LIN {X -172.185,Y +1147.423,Z +0.000,A -19.971,E1 -36.175,E3 +84213.761,E4 +0.000} C_DIS
LIN {X -165.999,Y +1152.127,Z +0.000,A -20.000,E1 -32.027,E3 +84233.519,E4 +0.000} C_DIS
LIN {X -160.138,Y +1155.667,Z +0.000,A -20.000,E1 -26.368,E3 +84257.889,E4 +0.000} C_DIS
LIN {X -155.625,Y +1157.756,Z +0.000,A -20.000,E1 -19.505,E3 +84286.565,E4 +0.000} C_DIS
LIN {X -153.552,Y +1158.113,Z +0.000,A -20.000,E1 -11.113,E3 +84322.316,E4 +0.000} C_DIS
LIN {X -156.311,Y +1155.540,Z +0.000,A -20.000,E1 -0.839,E3 +84365.676,E4 +0.000} C_DIS
LIN {X -161.281,Y +1151.851,Z +0.000,A -20.000,E1 +7.737,E3 +84395.575,E4 +0.000} C_DIS
LIN {X -167.493,Y +1147.157,Z +0.000,A -20.000,E1 +16.195,E3 +84420.014,E4 +0.000} C_DIS
LIN {X -173.235,Y +1142.221,Z +0.000,A -20.000,E1 +22.930,E3 +84437.316,E4 +0.000} C_DIS
LIN {X -181.123,Y +1133.734,Z +0.000,A -20.000,E1 +30.868,E3 +84458.072,E4 +0.000} C_DIS
LIN {X -189.654,Y +1120.856,Z +0.000,A -20.000,E1 +39.018,E3 +84480.086,E4 +0.000} C_DIS
LIN {X -195.246,Y +1107.046,Z +0.000,A -20.000,E1 +44.515,E3 +84497.988,E4 +0.000} C_DIS
LIN {X -198.051,Y +1092.368,Z +0.000,A -20.000,E1 +47.947,E3 +84514.514,E4 +0.000} C_DIS
LIN {X -198.143,Y +1081.370,Z +0.000,A -19.806,E1 +49.153,E3 +84526.375,E4 +0.000} C_DIS
LIN {X -197.177,Y +1073.569,Z +0.000,A -17.356,E1 +49.162,E3 +84534.959,E4 +0.000} C_DIS
LIN {X -195.448,Y +1066.139,Z +0.000,A -12.154,E1 +48.512,E3 +84543.554,E4 +0.000} C_DIS
LIN {X -193.346,Y +1058.941,Z +0.000,A -7.133,E1 +47.724,E3 +84552.434,E4 +0.000} C_DIS
LIN {X -191.781,Y +1050.839,Z +0.000,A -3.715,E1 +47.274,E3 +84562.767,E4 +0.000} C_DIS
LIN {X -190.795,Y +1039.355,Z +0.000,A -0.983,E1 +46.842,E3 +84577.427,E4 +0.000} C_DIS
LIN {X -190.395,Y +1028.856,Z +0.000,A -0.089,E1 +46.598,E3 +84590.821,E4 +0.000} C_DIS
LIN {X -190.239,Y +1018.851,Z +0.000,A -0.004,E1 +46.529,E3 +84603.589,E4 +0.000} C_DIS
LIN {X -190.161,Y +1004.975,Z +0.000,A +0.000,E1 +46.506,E3 +84621.303,E4 +0.000} C_DIS
LIN {X -190.142,Y +412.853,Z +0.000,A +0.000,E1 +46.501,E3 +85377.509,E4 +0.000} C_DIS
LIN {X -190.147,Y +401.077,Z +0.000,A +0.000,E1 +46.499,E3 +85392.550,E4 +0.000} C_DIS
LIN {X -190.159,Y +390.929,Z +0.000,A +0.000,E1 +46.494,E3 +85405.516,E4 +0.000} C_DIS
LIN {X -190.174,Y +383.973,Z +0.000,A +0.000,E1 +46.484,E3 +85414.409,E4 +0.000} C_DIS
LIN {X -190.200,Y +373.815,Z +0.000,A +0.000,E1 +46.448,E3 +85427.414,E4 +0.000} C_DIS
LIN {X -190.154,Y +361.003,Z +0.000,A +0.000,E1 +46.303,E3 +85443.908,E4 +0.000} C_DIS
LIN {X -189.772,Y +350.660,Z +0.000,A +0.049,E1 +45.996,E3 +85457.447,E4 +0.000} C_DIS
LIN {X -189.325,Y +346.917,Z +0.000,A +0.243,E1 +45.771,E3 +85462.516,E4 +0.000} C_DIS
LIN {X -188.196,Y +342.754,Z +0.000,A +1.966,E1 +45.249,E3 +85468.524,E4 +0.000} C_DIS
LIN {X -185.199,Y +337.023,Z +0.000,A +6.630,E1 +43.793,E3 +85477.898,E4 +0.000} C_DIS
LIN {X -181.141,Y +331.596,Z +0.000,A +12.274,E1 +41.569,E3 +85488.458,E4 +0.000} C_DIS
LIN {X -176.762,Y +326.804,Z +0.000,A +17.560,E1 +38.898,E3 +85499.882,E4 +0.000} C_DIS
LIN {X -172.184,Y +322.578,Z +0.000,A +19.859,E1 +36.197,E3 +85512.612,E4 +0.000} C_DIS
LIN {X -165.998,Y +317.874,Z +0.000,A +20.000,E1 +32.027,E3 +85532.370,E4 +0.000} C_DIS
LIN {X -160.137,Y +314.334,Z +0.000,A +20.000,E1 +26.368,E3 +85556.739,E4 +0.000} C_DIS
LIN {X -155.624,Y +312.245,Z +0.000,A +20.000,E1 +19.506,E3 +85585.415,E4 +0.000} C_DIS
LIN {X -153.557,Y +311.879,Z +0.000,A +20.000,E1 +11.113,E3 +85621.170,E4 +0.000} C_DIS
LIN {X -155.320,Y +313.348,Z +0.000,A +20.000,E1 +3.401,E3 +85654.354,E4 +0.000} C_DIS
LIN {X -160.005,Y +315.804,Z +0.000,A +20.000,E1 -4.720,E3 +85684.732,E4 +0.000} C_DIS
LIN {X -164.504,Y +318.255,Z +0.000,A +20.000,E1 -10.663,E3 +85704.101,E4 +0.000} C_DIS
LIN {X -170.340,Y +322.684,Z +0.000,A +20.000,E1 -17.457,E3 +85724.133,E4 +0.000} C_DIS
LIN {X -175.568,Y +329.106,Z +0.000,A +20.000,E1 -24.747,E3 +85741.367,E4 +0.000} C_DIS
LIN {X -184.074,Y +340.065,Z +0.000,A +20.000,E1 -33.664,E3 +85764.307,E4 +0.000} C_DIS
LIN {X -190.779,Y +351.388,Z +0.000,A +20.000,E1 -40.083,E3 +85782.085,E4 +0.000} C_DIS
LIN {X -195.254,Y +362.955,Z +0.000,A +20.000,E1 -44.515,E3 +85796.838,E4 +0.000} C_DIS
LIN {X -197.754,Y +374.780,Z +0.000,A +20.000,E1 -47.450,E3 +85810.260,E4 +0.000} C_DIS
LIN {X -198.310,Y +383.215,Z +0.000,A +19.956,E1 -48.698,E3 +85819.384,E4 +0.000} C_DIS
LIN {X -197.912,Y +391.275,Z +0.000,A +18.601,E1 -49.158,E3 +85828.102,E4 +0.000} C_DIS
LIN {X -196.679,Y +398.944,Z +0.000,A +13.989,E1 -48.784,E3 +85836.656,E4 +0.000} C_DIS
LIN {X -194.742,Y +406.288,Z +0.000,A +8.476,E1 -48.001,E3 +85845.339,E4 +0.000} C_DIS
LIN {X -192.748,Y +413.472,Z +0.000,A +3.905,E1 -47.267,E3 +85854.349,E4 +0.000} C_DIS
LIN {X -191.781,Y +419.162,Z +0.000,A +1.739,E1 -46.975,E3 +85861.617,E4 +0.000} C_DIS
LIN {X -190.795,Y +430.646,Z +0.000,A +0.152,E1 -46.707,E3 +85876.278,E4 +0.000} C_DIS
LIN {X -190.395,Y +441.145,Z +0.000,A +0.001,E1 -46.583,E3 +85889.671,E4 +0.000} C_DIS
LIN {X -190.239,Y +451.150,Z +0.000,A -0.000,E1 -46.528,E3 +85902.439,E4 +0.000} C_DIS
LIN {X -190.161,Y +465.026,Z +0.000,A -0.000,E1 -46.506,E3 +85920.154,E4 +0.000} C_DIS
LIN {X -190.142,Y +1057.148,Z +0.000,A -0.000,E1 -46.500,E3 +86676.360,E4 +0.000} C_DIS
LIN {X -190.147,Y +1068.924,Z +0.000,A -0.000,E1 -46.499,E3 +86691.401,E4 +0.000} C_DIS
LIN {X -190.159,Y +1079.072,Z +0.000,A -0.000,E1 -46.493,E3 +86704.366,E4 +0.000} C_DIS
LIN {X -190.174,Y +1086.028,Z +0.000,A -0.000,E1 -46.483,E3 +86713.260,E4 +0.000} C_DIS
LIN {X -190.200,Y +1096.186,Z +0.000,A -0.000,E1 -46.448,E3 +86726.264,E4 +0.000} C_DIS
LIN {X -190.154,Y +1108.998,Z +0.000,A -0.054,E1 -46.295,E3 +86742.759,E4 +0.000} C_DIS
LIN {X -189.772,Y +1119.341,Z +0.000,A -0.752,E1 -45.902,E3 +86756.297,E4 +0.000} C_DIS
LIN {X -189.097,Y +1124.276,Z +0.000,A -2.508,E1 -45.397,E3 +86763.029,E4 +0.000} C_DIS
LIN {X -187.410,Y +1129.069,Z +0.000,A -5.304,E1 -44.585,E3 +86770.202,E4 +0.000} C_DIS
LIN {X -183.899,Y +1134.873,Z +0.000,A -10.372,E1 -42.805,E3 +86780.208,E4 +0.000} C_DIS
LIN {X -179.711,Y +1140.065,Z +0.000,A -15.940,E1 -40.393,E3 +86790.994,E4 +0.000} C_DIS
LIN {X -176.763,Y +1143.197,Z +0.000,A -18.748,E1 -38.674,E3 +86798.732,E4 +0.000} C_DIS
LIN {X -172.185,Y +1147.423,Z +0.000,A -19.971,E1 -36.175,E3 +86811.462,E4 +0.000} C_DIS
LIN {X -165.999,Y +1152.127,Z +0.000,A -20.000,E1 -32.027,E3 +86831.220,E4 +0.000} C_DIS
LIN {X -160.138,Y +1155.667,Z +0.000,A -20.000,E1 -26.368,E3 +86855.590,E4 +0.000} C_DIS
LIN {X -155.625,Y +1157.756,Z +0.000,A -20.000,E1 -19.505,E3 +86884.266,E4 +0.000} C_DIS
LIN {X -153.552,Y +1158.113,Z +0.000,A -20.000,E1 -11.113,E3 +86920.017,E4 +0.000} C_DIS
LIN {X -156.311,Y +1155.540,Z +0.000,A -20.000,E1 -0.839,E3 +86963.377,E4 +0.000} C_DIS
LIN {X -161.281,Y +1151.851,Z +0.000,A -20.000,E1 +7.737,E3 +86993.276,E4 +0.000} C_DIS
LIN {X -167.493,Y +1147.157,Z +0.000,A -20.000,E1 +16.195,E3 +87017.715,E4 +0.000} C_DIS
LIN {X -173.235,Y +1142.221,Z +0.000,A -20.000,E1 +22.930,E3 +87035.017,E4 +0.000} C_DIS
LIN {X -181.123,Y +1133.734,Z +0.000,A -20.000,E1 +30.868,E3 +87055.773,E4 +0.000} C_DIS
LIN {X -189.654,Y +1120.856,Z +0.000,A -20.000,E1 +39.018,E3 +87077.787,E4 +0.000} C_DIS
LIN {X -195.246,Y +1107.046,Z +0.000,A -20.000,E1 +44.515,E3 +87095.689,E4 +0.000} C_DIS
LIN {X -198.051,Y +1092.368,Z +0.000,A -20.000,E1 +47.947,E3 +87112.215,E4 +0.000} C_DIS
LIN {X -198.143,Y +1081.370,Z +0.000,A -19.806,E1 +49.153,E3 +87124.076,E4 +0.000} C_DIS
LIN {X -197.177,Y +1073.569,Z +0.000,A -17.356,E1 +49.162,E3 +87132.660,E4 +0.000} C_DIS
LIN {X -195.448,Y +1066.139,Z +0.000,A -12.154,E1 +48.512,E3 +87141.255,E4 +0.000} C_DIS
LIN {X -193.346,Y +1058.941,Z +0.000,A -7.133,E1 +47.724,E3 +87150.135,E4 +0.000} C_DIS
LIN {X -191.781,Y +1050.839,Z +0.000,A -3.715,E1 +47.274,E3 +87160.468,E4 +0.000} C_DIS
LIN {X -190.795,Y +1039.355,Z +0.000,A -0.983,E1 +46.842,E3 +87175.128,E4 +0.000} C_DIS
LIN {X -190.395,Y +1028.856,Z +0.000,A -0.089,E1 +46.598,E3 +87188.522,E4 +0.000} C_DIS
LIN {X -190.239,Y +1018.851,Z +0.000,A -0.004,E1 +46.529,E3 +87201.290,E4 +0.000} C_DIS
LIN {X -190.161,Y +1004.975,Z +0.000,A +0.000,E1 +46.506,E3 +87219.004,E4 +0.000} C_DIS
LIN {X -190.142,Y +412.853,Z +0.000,A +0.000,E1 +46.501,E3 +87975.210,E4 +0.000} C_DIS
LIN {X -190.147,Y +401.077,Z +0.000,A +0.000,E1 +46.499,E3 +87990.251,E4 +0.000} C_DIS
LIN {X -190.159,Y +390.929,Z +0.000,A +0.000,E1 +46.494,E3 +88003.217,E4 +0.000} C_DIS
LIN {X -190.174,Y +383.973,Z +0.000,A +0.000,E1 +46.484,E3 +88012.110,E4 +0.000} C_DIS
LIN {X -190.200,Y +373.815,Z +0.000,A +0.000,E1 +46.448,E3 +88025.115,E4 +0.000} C_DIS
LIN {X -190.154,Y +361.003,Z +0.000,A +0.000,E1 +46.303,E3 +88041.609,E4 +0.000} C_DIS
LIN {X -189.772,Y +350.660,Z +0.000,A +0.049,E1 +45.996,E3 +88055.148,E4 +0.000} C_DIS
LIN {X -189.325,Y +346.917,Z +0.000,A +0.243,E1 +45.771,E3 +88060.217,E4 +0.000} C_DIS
LIN {X -188.196,Y +342.754,Z +0.000,A +1.966,E1 +45.249,E3 +88066.225,E4 +0.000} C_DIS
LIN {X -185.199,Y +337.023,Z +0.000,A +6.630,E1 +43.793,E3 +88075.599,E4 +0.000} C_DIS
LIN {X -181.141,Y +331.596,Z +0.000,A +12.274,E1 +41.569,E3 +88086.159,E4 +0.000} C_DIS
LIN {X -176.762,Y +326.804,Z +0.000,A +17.560,E1 +38.898,E3 +88097.583,E4 +0.000} C_DIS
LIN {X -172.184,Y +322.578,Z +0.000,A +19.859,E1 +36.197,E3 +88110.313,E4 +0.000} C_DIS
LIN {X -165.998,Y +317.874,Z +0.000,A +20.000,E1 +32.027,E3 +88130.071,E4 +0.000} C_DIS
LIN {X -160.137,Y +314.334,Z +0.000,A +20.000,E1 +26.368,E3 +88154.440,E4 +0.000} C_DIS
LIN {X -155.624,Y +312.245,Z +0.000,A +20.000,E1 +19.506,E3 +88183.116,E4 +0.000} C_DIS
LIN {X -153.557,Y +311.879,Z +0.000,A +20.000,E1 +11.113,E3 +88218.871,E4 +0.000} C_DIS
LIN {X -155.320,Y +313.348,Z +0.000,A +20.000,E1 +3.401,E3 +88252.055,E4 +0.000} C_DIS
LIN {X -160.005,Y +315.804,Z +0.000,A +20.000,E1 -4.720,E3 +88282.433,E4 +0.000} C_DIS
LIN {X -164.504,Y +318.255,Z +0.000,A +20.000,E1 -10.663,E3 +88301.802,E4 +0.000} C_DIS
LIN {X -170.340,Y +322.684,Z +0.000,A +20.000,E1 -17.457,E3 +88321.834,E4 +0.000} C_DIS
LIN {X -175.568,Y +329.106,Z +0.000,A +20.000,E1 -24.747,E3 +88339.068,E4 +0.000} C_DIS
LIN {X -184.074,Y +340.065,Z +0.000,A +20.000,E1 -33.664,E3 +88362.008,E4 +0.000} C_DIS
LIN {X -190.779,Y +351.388,Z +0.000,A +20.000,E1 -40.083,E3 +88379.786,E4 +0.000} C_DIS
LIN {X -195.254,Y +362.955,Z +0.000,A +20.000,E1 -44.515,E3 +88394.539,E4 +0.000} C_DIS
LIN {X -197.754,Y +374.780,Z +0.000,A +20.000,E1 -47.450,E3 +88407.961,E4 +0.000} C_DIS
LIN {X -198.310,Y +383.215,Z +0.000,A +19.956,E1 -48.698,E3 +88417.085,E4 +0.000} C_DIS
LIN {X -197.912,Y +391.275,Z +0.000,A +18.601,E1 -49.158,E3 +88425.803,E4 +0.000} C_DIS
LIN {X -196.679,Y +398.944,Z +0.000,A +13.989,E1 -48.784,E3 +88434.357,E4 +0.000} C_DIS
LIN {X -194.742,Y +406.288,Z +0.000,A +8.476,E1 -48.001,E3 +88443.040,E4 +0.000} C_DIS
LIN {X -192.748,Y +413.472,Z +0.000,A +3.905,E1 -47.267,E3 +88452.050,E4 +0.000} C_DIS
LIN {X -191.781,Y +419.162,Z +0.000,A +1.739,E1 -46.975,E3 +88459.318,E4 +0.000} C_DIS
LIN {X -190.795,Y +430.646,Z +0.000,A +0.152,E1 -46.707,E3 +88473.979,E4 +0.000} C_DIS
LIN {X -190.395,Y +441.145,Z +0.000,A +0.001,E1 -46.583,E3 +88487.372,E4 +0.000} C_DIS
LIN {X -190.239,Y +451.150,Z +0.000,A -0.000,E1 -46.528,E3 +88500.140,E4 +0.000} C_DIS
LIN {X -190.161,Y +465.026,Z +0.000,A -0.000,E1 -46.506,E3 +88517.855,E4 +0.000} C_DIS
LIN {X -190.142,Y +1057.148,Z +0.000,A -0.000,E1 -46.500,E3 +89274.061,E4 +0.000} C_DIS
LIN {X -190.147,Y +1068.924,Z +0.000,A -0.000,E1 -46.499,E3 +89289.102,E4 +0.000} C_DIS
LIN {X -190.159,Y +1079.072,Z +0.000,A -0.000,E1 -46.493,E3 +89302.067,E4 +0.000} C_DIS
LIN {X -190.174,Y +1086.028,Z +0.000,A -0.000,E1 -46.483,E3 +89310.961,E4 +0.000} C_DIS
LIN {X -190.200,Y +1096.186,Z +0.000,A -0.000,E1 -46.448,E3 +89323.965,E4 +0.000} C_DIS
LIN {X -190.154,Y +1108.998,Z +0.000,A -0.054,E1 -46.295,E3 +89340.460,E4 +0.000} C_DIS
LIN {X -189.772,Y +1119.341,Z +0.000,A -0.752,E1 -45.902,E3 +89353.998,E4 +0.000} C_DIS
LIN {X -189.097,Y +1124.276,Z +0.000,A -2.508,E1 -45.397,E3 +89360.730,E4 +0.000} C_DIS
LIN {X -187.410,Y +1129.069,Z +0.000,A -5.304,E1 -44.585,E3 +89367.903,E4 +0.000} C_DIS
LIN {X -183.899,Y +1134.873,Z +0.000,A -10.372,E1 -42.805,E3 +89377.909,E4 +0.000} C_DIS
LIN {X -179.711,Y +1140.065,Z +0.000,A -15.940,E1 -40.393,E3 +89388.695,E4 +0.000} C_DIS
LIN {X -176.763,Y +1143.197,Z +0.000,A -18.748,E1 -38.674,E3 +89396.433,E4 +0.000} C_DIS
LIN {X -172.185,Y +1147.423,Z +0.000,A -19.971,E1 -36.175,E3 +89409.163,E4 +0.000} C_DIS
LIN {X -165.999,Y +1152.127,Z +0.000,A -20.000,E1 -32.027,E3 +89428.921,E4 +0.000} C_DIS
LIN {X -160.138,Y +1155.667,Z +0.000,A -20.000,E1 -26.368,E3 +89453.291,E4 +0.000} C_DIS
LIN {X -155.625,Y +1157.756,Z +0.000,A -20.000,E1 -19.505,E3 +89481.967,E4 +0.000} C_DIS
LIN {X -153.552,Y +1158.113,Z +0.000,A -20.000,E1 -11.113,E3 +89517.718,E4 +0.000} C_DIS
LIN {X -156.311,Y +1155.540,Z +0.000,A -20.000,E1 -0.839,E3 +89561.078,E4 +0.000} C_DIS
LIN {X -161.281,Y +1151.851,Z +0.000,A -20.000,E1 +7.737,E3 +89590.977,E4 +0.000} C_DIS
LIN {X -167.493,Y +1147.157,Z +0.000,A -20.000,E1 +16.195,E3 +89615.416,E4 +0.000} C_DIS
LIN {X -173.235,Y +1142.221,Z +0.000,A -20.000,E1 +22.930,E3 +89632.718,E4 +0.000} C_DIS
LIN {X -181.123,Y +1133.734,Z +0.000,A -20.000,E1 +30.868,E3 +89653.474,E4 +0.000} C_DIS
LIN {X -189.654,Y +1120.856,Z +0.000,A -20.000,E1 +39.018,E3 +89675.488,E4 +0.000} C_DIS
LIN {X -195.246,Y +1107.046,Z +0.000,A -20.000,E1 +44.515,E3 +89693.390,E4 +0.000} C_DIS
LIN {X -198.051,Y +1092.368,Z +0.000,A -20.000,E1 +47.947,E3 +89709.916,E4 +0.000} C_DIS
LIN {X -198.143,Y +1081.370,Z +0.000,A -19.806,E1 +49.153,E3 +89721.777,E4 +0.000} C_DIS
LIN {X -197.177,Y +1073.569,Z +0.000,A -17.356,E1 +49.162,E3 +89730.361,E4 +0.000} C_DIS
LIN {X -195.448,Y +1066.139,Z +0.000,A -12.154,E1 +48.512,E3 +89738.956,E4 +0.000} C_DIS
LIN {X -193.346,Y +1058.941,Z +0.000,A -7.133,E1 +47.724,E3 +89747.836,E4 +0.000} C_DIS
LIN {X -191.781,Y +1050.839,Z +0.000,A -3.715,E1 +47.274,E3 +89758.169,E4 +0.000} C_DIS
LIN {X -190.795,Y +1039.355,Z +0.000,A -0.983,E1 +46.842,E3 +89772.829,E4 +0.000} C_DIS
LIN {X -190.395,Y +1028.856,Z +0.000,A -0.089,E1 +46.598,E3 +89786.223,E4 +0.000} C_DIS
LIN {X -190.239,Y +1018.851,Z +0.000,A -0.004,E1 +46.529,E3 +89798.991,E4 +0.000} C_DIS
LIN {X -190.161,Y +1004.975,Z +0.000,A +0.000,E1 +46.506,E3 +89816.705,E4 +0.000} C_DIS
LIN {X -190.142,Y +412.853,Z +0.000,A +0.000,E1 +46.501,E3 +90572.911,E4 +0.000} C_DIS
LIN {X -190.147,Y +401.077,Z +0.000,A +0.000,E1 +46.499,E3 +90587.952,E4 +0.000} C_DIS
LIN {X -190.159,Y +390.929,Z +0.000,A +0.000,E1 +46.494,E3 +90600.918,E4 +0.000} C_DIS
LIN {X -190.174,Y +383.973,Z +0.000,A +0.000,E1 +46.484,E3 +90609.811,E4 +0.000} C_DIS
LIN {X -190.200,Y +373.815,Z +0.000,A +0.000,E1 +46.448,E3 +90622.816,E4 +0.000} C_DIS
LIN {X -190.154,Y +361.003,Z +0.000,A +0.000,E1 +46.303,E3 +90639.310,E4 +0.000} C_DIS
LIN {X -189.772,Y +350.660,Z +0.000,A +0.049,E1 +45.996,E3 +90652.849,E4 +0.000} C_DIS
LIN {X -189.325,Y +346.917,Z +0.000,A +0.243,E1 +45.771,E3 +90657.918,E4 +0.000} C_DIS
LIN {X -188.196,Y +342.754,Z +0.000,A +1.966,E1 +45.249,E3 +90663.926,E4 +0.000} C_DIS
LIN {X -185.199,Y +337.023,Z +0.000,A +6.630,E1 +43.793,E3 +90673.300,E4 +0.000} C_DIS
LIN {X -181.141,Y +331.596,Z +0.000,A +12.274,E1 +41.569,E3 +90683.860,E4 +0.000} C_DIS
LIN {X -176.762,Y +326.804,Z +0.000,A +17.560,E1 +38.898,E3 +90695.284,E4 +0.000} C_DIS
LIN {X -172.184,Y +322.578,Z +0.000,A +19.859,E1 +36.197,E3 +90708.014,E4 +0.000} C_DIS
LIN {X -165.998,Y +317.874,Z +0.000,A +20.000,E1 +32.027,E3 +90727.772,E4 +0.000} C_DIS
LIN {X -160.137,Y +314.334,Z +0.000,A +20.000,E1 +26.368,E3 +90752.141,E4 +0.000} C_DIS
LIN {X -155.624,Y +312.245,Z +0.000,A +20.000,E1 +19.506,E3 +90780.817,E4 +0.000} C_DIS
LIN {X -153.557,Y +311.879,Z +0.000,A +20.000,E1 +11.113,E3 +90816.572,E4 +0.000} C_DIS
LIN {X -155.320,Y +313.348,Z +0.000,A +20.000,E1 +3.401,E3 +90849.756,E4 +0.000} C_DIS
LIN {X -160.005,Y +315.804,Z +0.000,A +20.000,E1 -4.720,E3 +90880.134,E4 +0.000} C_DIS
LIN {X -164.504,Y +318.255,Z +0.000,A +20.000,E1 -10.663,E3 +90899.503,E4 +0.000} C_DIS
LIN {X -170.340,Y +322.684,Z +0.000,A +20.000,E1 -17.457,E3 +90919.535,E4 +0.000} C_DIS
LIN {X -175.568,Y +329.106,Z +0.000,A +20.000,E1 -24.747,E3 +90936.769,E4 +0.000} C_DIS
LIN {X -184.074,Y +340.065,Z +0.000,A +20.000,E1 -33.664,E3 +90959.709,E4 +0.000} C_DIS
LIN {X -190.779,Y +351.388,Z +0.000,A +20.000,E1 -40.083,E3 +90977.487,E4 +0.000} C_DIS
LIN {X -195.254,Y +362.955,Z +0.000,A +20.000,E1 -44.515,E3 +90992.240,E4 +0.000} C_DIS
LIN {X -197.754,Y +374.780,Z +0.000,A +20.000,E1 -47.450,E3 +91005.662,E4 +0.000} C_DIS
LIN {X -198.310,Y +383.215,Z +0.000,A +19.956,E1 -48.698,E3 +91014.786,E4 +0.000} C_DIS
LIN {X -197.912,Y +391.275,Z +0.000,A +18.601,E1 -49.158,E3 +91023.504,E4 +0.000} C_DIS
LIN {X -196.679,Y +398.944,Z +0.000,A +13.989,E1 -48.784,E3 +91032.058,E4 +0.000} C_DIS
LIN {X -194.742,Y +406.288,Z +0.000,A +8.476,E1 -48.001,E3 +91040.741,E4 +0.000} C_DIS
LIN {X -192.748,Y +413.472,Z +0.000,A +3.905,E1 -47.267,E3 +91049.751,E4 +0.000} C_DIS
LIN {X -191.781,Y +419.162,Z +0.000,A +1.739,E1 -46.975,E3 +91057.019,E4 +0.000} C_DIS
LIN {X -190.795,Y +430.646,Z +0.000,A +0.152,E1 -46.707,E3 +91071.680,E4 +0.000} C_DIS
LIN {X -190.395,Y +441.145,Z +0.000,A +0.001,E1 -46.583,E3 +91085.073,E4 +0.000} C_DIS
LIN {X -190.239,Y +451.150,Z +0.000,A -0.000,E1 -46.528,E3 +91097.841,E4 +0.000} C_DIS
LIN {X -190.161,Y +465.026,Z +0.000,A -0.000,E1 -46.506,E3 +91115.556,E4 +0.000} C_DIS
LIN {X -190.142,Y +1057.148,Z +0.000,A -0.000,E1 -46.500,E3 +91871.762,E4 +0.000} C_DIS
LIN {X -190.147,Y +1068.924,Z +0.000,A -0.000,E1 -46.499,E3 +91886.803,E4 +0.000} C_DIS
LIN {X -190.159,Y +1079.072,Z +0.000,A -0.000,E1 -46.493,E3 +91899.768,E4 +0.000} C_DIS
LIN {X -190.174,Y +1086.028,Z +0.000,A -0.000,E1 -46.483,E3 +91908.662,E4 +0.000} C_DIS
LIN {X -190.200,Y +1096.186,Z +0.000,A -0.000,E1 -46.448,E3 +91921.666,E4 +0.000} C_DIS
LIN {X -190.154,Y +1108.998,Z +0.000,A -0.054,E1 -46.295,E3 +91938.161,E4 +0.000} C_DIS
LIN {X -189.772,Y +1119.341,Z +0.000,A -0.752,E1 -45.902,E3 +91951.699,E4 +0.000} C_DIS
LIN {X -189.097,Y +1124.276,Z +0.000,A -2.508,E1 -45.397,E3 +91958.431,E4 +0.000} C_DIS
LIN {X -187.410,Y +1129.069,Z +0.000,A -5.304,E1 -44.585,E3 +91965.604,E4 +0.000} C_DIS
LIN {X -183.899,Y +1134.873,Z +0.000,A -10.372,E1 -42.805,E3 +91975.610,E4 +0.000} C_DIS
LIN {X -179.711,Y +1140.065,Z +0.000,A -15.940,E1 -40.393,E3 +91986.396,E4 +0.000} C_DIS
LIN {X -176.763,Y +1143.197,Z +0.000,A -18.748,E1 -38.674,E3 +91994.134,E4 +0.000} C_DIS
LIN {X -172.185,Y +1147.423,Z +0.000,A -19.971,E1 -36.175,E3 +92006.864,E4 +0.000} C_DIS
LIN {X -165.999,Y +1152.127,Z +0.000,A -20.000,E1 -32.027,E3 +92026.622,E4 +0.000} C_DIS
LIN {X -160.138,Y +1155.667,Z +0.000,A -20.000,E1 -26.368,E3 +92050.992,E4 +0.000} C_DIS
LIN {X -155.625,Y +1157.756,Z +0.000,A -20.000,E1 -19.505,E3 +92079.668,E4 +0.000} C_DIS
LIN {X -153.552,Y +1158.113,Z +0.000,A -20.000,E1 -11.113,E3 +92115.419,E4 +0.000} C_DIS
LIN {X -156.311,Y +1155.540,Z +0.000,A -20.000,E1 -0.839,E3 +92158.779,E4 +0.000} C_DIS
LIN {X -161.281,Y +1151.851,Z +0.000,A -20.000,E1 +7.737,E3 +92188.678,E4 +0.000} C_DIS
LIN {X -167.493,Y +1147.157,Z +0.000,A -20.000,E1 +16.195,E3 +92213.117,E4 +0.000} C_DIS
LIN {X -173.235,Y +1142.221,Z +0.000,A -20.000,E1 +22.930,E3 +92230.419,E4 +0.000} C_DIS
LIN {X -181.123,Y +1133.734,Z +0.000,A -20.000,E1 +30.868,E3 +92251.175,E4 +0.000} C_DIS
LIN {X -189.654,Y +1120.856,Z +0.000,A -20.000,E1 +39.018,E3 +92273.189,E4 +0.000} C_DIS
LIN {X -195.246,Y +1107.046,Z +0.000,A -20.000,E1 +44.515,E3 +92291.091,E4 +0.000} C_DIS
LIN {X -198.051,Y +1092.368,Z +0.000,A -20.000,E1 +47.947,E3 +92307.617,E4 +0.000} C_DIS
LIN {X -198.143,Y +1081.370,Z +0.000,A -19.806,E1 +49.153,E3 +92319.478,E4 +0.000} C_DIS
LIN {X -197.177,Y +1073.569,Z +0.000,A -17.356,E1 +49.162,E3 +92328.062,E4 +0.000} C_DIS
LIN {X -195.448,Y +1066.139,Z +0.000,A -12.154,E1 +48.512,E3 +92336.657,E4 +0.000} C_DIS
LIN {X -193.346,Y +1058.941,Z +0.000,A -7.133,E1 +47.724,E3 +92345.537,E4 +0.000} C_DIS
LIN {X -191.781,Y +1050.839,Z +0.000,A -3.715,E1 +47.274,E3 +92355.870,E4 +0.000} C_DIS
LIN {X -190.795,Y +1039.355,Z +0.000,A -0.983,E1 +46.842,E3 +92370.530,E4 +0.000} C_DIS
LIN {X -190.395,Y +1028.856,Z +0.000,A -0.089,E1 +46.598,E3 +92383.924,E4 +0.000} C_DIS
LIN {X -190.239,Y +1018.851,Z +0.000,A -0.004,E1 +46.529,E3 +92396.692,E4 +0.000} C_DIS
LIN {X -190.161,Y +1004.975,Z +0.000,A +0.000,E1 +46.506,E3 +92414.406,E4 +0.000} C_DIS
LIN {X -190.142,Y +412.853,Z +0.000,A +0.000,E1 +46.501,E3 +93170.612,E4 +0.000} C_DIS
LIN {X -190.147,Y +401.077,Z +0.000,A +0.000,E1 +46.499,E3 +93185.653,E4 +0.000} C_DIS
LIN {X -190.159,Y +390.929,Z +0.000,A +0.000,E1 +46.494,E3 +93198.619,E4 +0.000} C_DIS
LIN {X -190.174,Y +383.973,Z +0.000,A +0.000,E1 +46.484,E3 +93207.512,E4 +0.000} C_DIS
LIN {X -190.200,Y +373.815,Z +0.000,A +0.000,E1 +46.448,E3 +93220.517,E4 +0.000} C_DIS
LIN {X -190.154,Y +361.003,Z +0.000,A +0.000,E1 +46.303,E3 +93237.011,E4 +0.000} C_DIS
LIN {X -189.772,Y +350.660,Z +0.000,A +0.049,E1 +45.996,E3 +93250.550,E4 +0.000} C_DIS
LIN {X -189.325,Y +346.917,Z +0.000,A +0.243,E1 +45.771,E3 +93255.619,E4 +0.000} C_DIS
LIN {X -188.196,Y +342.754,Z +0.000,A +1.966,E1 +45.249,E3 +93261.627,E4 +0.000} C_DIS
LIN {X -185.199,Y +337.023,Z +0.000,A +6.630,E1 +43.793,E3 +93271.001,E4 +0.000} C_DIS
LIN {X -181.141,Y +331.596,Z +0.000,A +12.274,E1 +41.569,E3 +93281.561,E4 +0.000} C_DIS
LIN {X -176.762,Y +326.804,Z +0.000,A +17.560,E1 +38.898,E3 +93292.985,E4 +0.000} C_DIS
LIN {X -172.184,Y +322.578,Z +0.000,A +19.859,E1 +36.197,E3 +93305.715,E4 +0.000} C_DIS
LIN {X -165.998,Y +317.874,Z +0.000,A +20.000,E1 +32.027,E3 +93325.473,E4 +0.000} C_DIS
LIN {X -160.137,Y +314.334,Z +0.000,A +20.000,E1 +26.368,E3 +93349.842,E4 +0.000} C_DIS
LIN {X -155.624,Y +312.245,Z +0.000,A +20.000,E1 +19.506,E3 +93378.518,E4 +0.000} C_DIS
LIN {X -153.557,Y +311.879,Z +0.000,A +20.000,E1 +11.113,E3 +93414.273,E4 +0.000} C_DIS
LIN {X -155.320,Y +313.348,Z +0.000,A +20.000,E1 +3.401,E3 +93447.457,E4 +0.000} C_DIS
LIN {X -160.005,Y +315.804,Z +0.000,A +20.000,E1 -4.720,E3 +93477.835,E4 +0.000} C_DIS
LIN {X -164.504,Y +318.255,Z +0.000,A +20.000,E1 -10.663,E3 +93497.204,E4 +0.000} C_DIS
LIN {X -170.340,Y +322.684,Z +0.000,A +20.000,E1 -17.457,E3 +93517.236,E4 +0.000} C_DIS
LIN {X -175.568,Y +329.106,Z +0.000,A +20.000,E1 -24.747,E3 +93534.470,E4 +0.000} C_DIS
LIN {X -184.074,Y +340.065,Z +0.000,A +20.000,E1 -33.664,E3 +93557.410,E4 +0.000} C_DIS
LIN {X -190.779,Y +351.388,Z +0.000,A +20.000,E1 -40.083,E3 +93575.188,E4 +0.000} C_DIS
LIN {X -195.254,Y +362.955,Z +0.000,A +20.000,E1 -44.515,E3 +93589.941,E4 +0.000} C_DIS
LIN {X -197.754,Y +374.780,Z +0.000,A +20.000,E1 -47.450,E3 +93603.363,E4 +0.000} C_DIS
LIN {X -198.310,Y +383.215,Z +0.000,A +19.956,E1 -48.698,E3 +93612.487,E4 +0.000} C_DIS
LIN {X -197.912,Y +391.275,Z +0.000,A +18.601,E1 -49.158,E3 +93621.205,E4 +0.000} C_DIS
LIN {X -196.679,Y +398.944,Z +0.000,A +13.989,E1 -48.784,E3 +93629.759,E4 +0.000} C_DIS
LIN {X -194.742,Y +406.288,Z +0.000,A +8.476,E1 -48.001,E3 +93638.442,E4 +0.000} C_DIS
LIN {X -192.748,Y +413.472,Z +0.000,A +3.905,E1 -47.267,E3 +93647.452,E4 +0.000} C_DIS
LIN {X -191.781,Y +419.162,Z +0.000,A +1.739,E1 -46.975,E3 +93654.720,E4 +0.000} C_DIS
LIN {X -190.795,Y +430.646,Z +0.000,A +0.152,E1 -46.707,E3 +93669.381,E4 +0.000} C_DIS
LIN {X -190.395,Y +441.145,Z +0.000,A +0.001,E1 -46.583,E3 +93682.774,E4 +0.000} C_DIS
LIN {X -190.239,Y +451.150,Z +0.000,A -0.000,E1 -46.528,E3 +93695.542,E4 +0.000} C_DIS
LIN {X -190.161,Y +465.026,Z +0.000,A -0.000,E1 -46.506,E3 +93713.257,E4 +0.000} C_DIS
LIN {X -190.142,Y +1057.148,Z +0.000,A -0.000,E1 -46.500,E3 +94469.463,E4 +0.000} C_DIS
LIN {X -190.147,Y +1068.924,Z +0.000,A -0.000,E1 -46.499,E3 +94484.504,E4 +0.000} C_DIS
LIN {X -190.159,Y +1079.072,Z +0.000,A -0.000,E1 -46.493,E3 +94497.469,E4 +0.000} C_DIS
LIN {X -190.174,Y +1086.028,Z +0.000,A -0.000,E1 -46.483,E3 +94506.363,E4 +0.000} C_DIS
LIN {X -190.200,Y +1096.186,Z +0.000,A -0.000,E1 -46.448,E3 +94519.367,E4 +0.000} C_DIS
LIN {X -190.154,Y +1108.998,Z +0.000,A -0.054,E1 -46.295,E3 +94535.862,E4 +0.000} C_DIS
LIN {X -189.772,Y +1119.341,Z +0.000,A -0.752,E1 -45.902,E3 +94549.400,E4 +0.000} C_DIS
LIN {X -189.097,Y +1124.276,Z +0.000,A -2.508,E1 -45.397,E3 +94556.132,E4 +0.000} C_DIS
LIN {X -187.410,Y +1129.069,Z +0.000,A -5.304,E1 -44.585,E3 +94563.305,E4 +0.000} C_DIS
LIN {X -183.899,Y +1134.873,Z +0.000,A -10.372,E1 -42.805,E3 +94573.311,E4 +0.000} C_DIS
LIN {X -179.711,Y +1140.065,Z +0.000,A -15.940,E1 -40.393,E3 +94584.097,E4 +0.000} C_DIS
LIN {X -176.763,Y +1143.197,Z +0.000,A -18.748,E1 -38.674,E3 +94591.835,E4 +0.000} C_DIS
LIN {X -172.185,Y +1147.423,Z +0.000,A -19.971,E1 -36.175,E3 +94604.565,E4 +0.000} C_DIS
LIN {X -165.999,Y +1152.127,Z +0.000,A -20.000,E1 -32.027,E3 +94624.323,E4 +0.000} C_DIS
LIN {X -160.138,Y +1155.667,Z +0.000,A -20.000,E1 -26.368,E3 +94648.693,E4 +0.000} C_DIS
LIN {X -155.625,Y +1157.756,Z +0.000,A -20.000,E1 -19.505,E3 +94677.369,E4 +0.000} C_DIS
LIN {X -153.552,Y +1158.113,Z +0.000,A -20.000,E1 -11.113,E3 +94713.120,E4 +0.000} C_DIS
LIN {X -156.311,Y +1155.540,Z +0.000,A -20.000,E1 -0.839,E3 +94756.480,E4 +0.000} C_DIS
LIN {X -161.281,Y +1151.851,Z +0.000,A -20.000,E1 +7.737,E3 +94786.379,E4 +0.000} C_DIS
LIN {X -167.493,Y +1147.157,Z +0.000,A -20.000,E1 +16.195,E3 +94810.818,E4 +0.000} C_DIS
LIN {X -173.235,Y +1142.221,Z +0.000,A -20.000,E1 +22.930,E3 +94828.120,E4 +0.000} C_DIS
LIN {X -181.123,Y +1133.734,Z +0.000,A -20.000,E1 +30.868,E3 +94848.876,E4 +0.000} C_DIS
LIN {X -189.654,Y +1120.856,Z +0.000,A -20.000,E1 +39.018,E3 +94870.890,E4 +0.000} C_DIS
LIN {X -195.246,Y +1107.046,Z +0.000,A -20.000,E1 +44.515,E3 +94888.792,E4 +0.000} C_DIS
LIN {X -198.051,Y +1092.368,Z +0.000,A -20.000,E1 +47.947,E3 +94905.318,E4 +0.000} C_DIS
LIN {X -198.143,Y +1081.370,Z +0.000,A -19.806,E1 +49.153,E3 +94917.179,E4 +0.000} C_DIS
LIN {X -197.177,Y +1073.569,Z +0.000,A -17.356,E1 +49.162,E3 +94925.763,E4 +0.000} C_DIS
LIN {X -195.448,Y +1066.139,Z +0.000,A -12.154,E1 +48.512,E3 +94934.358,E4 +0.000} C_DIS
LIN {X -193.346,Y +1058.941,Z +0.000,A -7.133,E1 +47.724,E3 +94943.238,E4 +0.000} C_DIS
LIN {X -191.781,Y +1050.839,Z +0.000,A -3.715,E1 +47.274,E3 +94953.571,E4 +0.000} C_DIS
LIN {X -190.795,Y +1039.355,Z +0.000,A -0.983,E1 +46.842,E3 +94968.231,E4 +0.000} C_DIS
LIN {X -190.395,Y +1028.856,Z +0.000,A -0.089,E1 +46.598,E3 +94981.625,E4 +0.000} C_DIS
LIN {X -190.239,Y +1018.851,Z +0.000,A -0.004,E1 +46.529,E3 +94994.393,E4 +0.000} C_DIS
LIN {X -190.161,Y +1004.975,Z +0.000,A +0.000,E1 +46.506,E3 +95012.107,E4 +0.000} C_DIS
LIN {X -190.142,Y +412.853,Z +0.000,A +0.000,E1 +46.501,E3 +95768.313,E4 +0.000} C_DIS
LIN {X -190.147,Y +401.077,Z +0.000,A +0.000,E1 +46.499,E3 +95783.354,E4 +0.000} C_DIS
LIN {X -190.159,Y +390.929,Z +0.000,A +0.000,E1 +46.494,E3 +95796.320,E4 +0.000} C_DIS
LIN {X -190.174,Y +383.973,Z +0.000,A +0.000,E1 +46.484,E3 +95805.213,E4 +0.000} C_DIS
LIN {X -190.200,Y +373.815,Z +0.000,A +0.000,E1 +46.448,E3 +95818.218,E4 +0.000} C_DIS
LIN {X -190.154,Y +361.003,Z +0.000,A +0.000,E1 +46.303,E3 +95834.712,E4 +0.000} C_DIS
LIN {X -189.772,Y +350.660,Z +0.000,A +0.049,E1 +45.996,E3 +95848.251,E4 +0.000} C_DIS
LIN {X -189.325,Y +346.917,Z +0.000,A +0.243,E1 +45.771,E3 +95853.320,E4 +0.000} C_DIS
LIN {X -188.196,Y +342.754,Z +0.000,A +1.966,E1 +45.249,E3 +95859.328,E4 +0.000} C_DIS
LIN {X -185.199,Y +337.023,Z +0.000,A +6.630,E1 +43.793,E3 +95868.702,E4 +0.000} C_DIS
LIN {X -181.141,Y +331.596,Z +0.000,A +12.274,E1 +41.569,E3 +95879.262,E4 +0.000} C_DIS
LIN {X -176.762,Y +326.804,Z +0.000,A +17.560,E1 +38.898,E3 +95890.686,E4 +0.000} C_DIS
LIN {X -172.184,Y +322.578,Z +0.000,A +19.859,E1 +36.197,E3 +95903.416,E4 +0.000} C_DIS
LIN {X -165.998,Y +317.874,Z +0.000,A +20.000,E1 +32.027,E3 +95923.174,E4 +0.000} C_DIS
LIN {X -160.137,Y +314.334,Z +0.000,A +20.000,E1 +26.368,E3 +95947.543,E4 +0.000} C_DIS
LIN {X -155.624,Y +312.245,Z +0.000,A +20.000,E1 +19.506,E3 +95976.219,E4 +0.000} C_DIS
LIN {X -153.557,Y +311.879,Z +0.000,A +20.000,E1 +11.113,E3 +96011.974,E4 +0.000} C_DIS
LIN {X -155.320,Y +313.348,Z +0.000,A +20.000,E1 +3.401,E3 +96045.158,E4 +0.000} C_DIS
LIN {X -160.005,Y +315.804,Z +0.000,A +20.000,E1 -4.720,E3 +96075.536,E4 +0.000} C_DIS
LIN {X -164.504,Y +318.255,Z +0.000,A +20.000,E1 -10.663,E3 +96094.905,E4 +0.000} C_DIS
LIN {X -170.340,Y +322.684,Z +0.000,A +20.000,E1 -17.457,E3 +96114.937,E4 +0.000} C_DIS
LIN {X -175.568,Y +329.106,Z +0.000,A +20.000,E1 -24.747,E3 +96132.171,E4 +0.000} C_DIS
LIN {X -184.074,Y +340.065,Z +0.000,A +20.000,E1 -33.664,E3 +96155.111,E4 +0.000} C_DIS
LIN {X -190.779,Y +351.388,Z +0.000,A +20.000,E1 -40.083,E3 +96172.889,E4 +0.000} C_DIS
LIN {X -195.254,Y +362.955,Z +0.000,A +20.000,E1 -44.515,E3 +96187.642,E4 +0.000} C_DIS
LIN {X -197.754,Y +374.780,Z +0.000,A +20.000,E1 -47.450,E3 +96201.064,E4 +0.000} C_DIS
LIN {X -198.310,Y +383.215,Z +0.000,A +19.956,E1 -48.698,E3 +96210.188,E4 +0.000} C_DIS
LIN {X -197.912,Y +391.275,Z +0.000,A +18.601,E1 -49.158,E3 +96218.906,E4 +0.000} C_DIS
LIN {X -196.679,Y +398.944,Z +0.000,A +13.989,E1 -48.784,E3 +96227.460,E4 +0.000} C_DIS
LIN {X -194.742,Y +406.288,Z +0.000,A +8.476,E1 -48.001,E3 +96236.143,E4 +0.000} C_DIS
LIN {X -192.748,Y +413.472,Z +0.000,A +3.905,E1 -47.267,E3 +96245.153,E4 +0.000} C_DIS
LIN {X -191.781,Y +419.162,Z +0.000,A +1.739,E1 -46.975,E3 +96252.421,E4 +0.000} C_DIS
LIN {X -190.795,Y +430.646,Z +0.000,A +0.152,E1 -46.707,E3 +96267.082,E4 +0.000} C_DIS
LIN {X -190.395,Y +441.145,Z +0.000,A +0.001,E1 -46.583,E3 +96280.475,E4 +0.000} C_DIS
LIN {X -190.239,Y +451.150,Z +0.000,A -0.000,E1 -46.528,E3 +96293.243,E4 +0.000} C_DIS
LIN {X -190.161,Y +465.026,Z +0.000,A -0.000,E1 -46.506,E3 +96310.958,E4 +0.000} C_DIS
LIN {X -190.142,Y +1057.148,Z +0.000,A -0.000,E1 -46.500,E3 +97067.164,E4 +0.000} C_DIS
LIN {X -190.147,Y +1068.924,Z +0.000,A -0.000,E1 -46.499,E3 +97082.205,E4 +0.000} C_DIS
LIN {X -190.159,Y +1079.072,Z +0.000,A -0.000,E1 -46.493,E3 +97095.170,E4 +0.000} C_DIS
LIN {X -190.174,Y +1086.028,Z +0.000,A -0.000,E1 -46.483,E3 +97104.064,E4 +0.000} C_DIS
LIN {X -190.200,Y +1096.186,Z +0.000,A -0.000,E1 -46.448,E3 +97117.068,E4 +0.000} C_DIS
LIN {X -190.154,Y +1108.998,Z +0.000,A -0.054,E1 -46.295,E3 +97133.563,E4 +0.000} C_DIS
LIN {X -189.772,Y +1119.341,Z +0.000,A -0.752,E1 -45.902,E3 +97147.101,E4 +0.000} C_DIS
LIN {X -189.097,Y +1124.276,Z +0.000,A -2.508,E1 -45.397,E3 +97153.833,E4 +0.000} C_DIS
LIN {X -187.410,Y +1129.069,Z +0.000,A -5.304,E1 -44.585,E3 +97161.006,E4 +0.000} C_DIS
LIN {X -183.899,Y +1134.873,Z +0.000,A -10.372,E1 -42.805,E3 +97171.012,E4 +0.000} C_DIS
LIN {X -179.711,Y +1140.065,Z +0.000,A -15.940,E1 -40.393,E3 +97181.798,E4 +0.000} C_DIS
LIN {X -176.763,Y +1143.197,Z +0.000,A -18.748,E1 -38.674,E3 +97189.536,E4 +0.000} C_DIS
LIN {X -172.185,Y +1147.423,Z +0.000,A -19.971,E1 -36.175,E3 +97202.266,E4 +0.000} C_DIS
LIN {X -165.999,Y +1152.127,Z +0.000,A -20.000,E1 -32.027,E3 +97222.024,E4 +0.000} C_DIS
LIN {X -160.138,Y +1155.667,Z +0.000,A -20.000,E1 -26.368,E3 +97246.394,E4 +0.000} C_DIS
LIN {X -155.625,Y +1157.756,Z +0.000,A -20.000,E1 -19.505,E3 +97275.070,E4 +0.000} C_DIS
LIN {X -153.552,Y +1158.113,Z +0.000,A -20.000,E1 -11.113,E3 +97310.821,E4 +0.000} C_DIS
LIN {X -156.311,Y +1155.540,Z +0.000,A -20.000,E1 -0.839,E3 +97354.181,E4 +0.000} C_DIS
LIN {X -161.281,Y +1151.851,Z +0.000,A -20.000,E1 +7.737,E3 +97384.080,E4 +0.000} C_DIS
LIN {X -167.493,Y +1147.157,Z +0.000,A -20.000,E1 +16.195,E3 +97408.519,E4 +0.000} C_DIS
LIN {X -173.235,Y +1142.221,Z +0.000,A -20.000,E1 +22.930,E3 +97425.821,E4 +0.000} C_DIS
LIN {X -181.123,Y +1133.734,Z +0.000,A -20.000,E1 +30.868,E3 +97446.577,E4 +0.000} C_DIS
LIN {X -189.654,Y +1120.856,Z +0.000,A -20.000,E1 +39.018,E3 +97468.591,E4 +0.000} C_DIS
LIN {X -195.246,Y +1107.046,Z +0.000,A -20.000,E1 +44.515,E3 +97486.493,E4 +0.000} C_DIS
LIN {X -198.051,Y +1092.368,Z +0.000,A -20.000,E1 +47.947,E3 +97503.019,E4 +0.000} C_DIS
LIN {X -198.143,Y +1081.370,Z +0.000,A -19.806,E1 +49.153,E3 +97514.880,E4 +0.000} C_DIS
LIN {X -197.177,Y +1073.569,Z +0.000,A -17.356,E1 +49.162,E3 +97523.464,E4 +0.000} C_DIS
LIN {X -195.448,Y +1066.139,Z +0.000,A -12.154,E1 +48.512,E3 +97532.059,E4 +0.000} C_DIS
LIN {X -193.346,Y +1058.941,Z +0.000,A -7.133,E1 +47.724,E3 +97540.939,E4 +0.000} C_DIS
LIN {X -191.781,Y +1050.839,Z +0.000,A -3.715,E1 +47.274,E3 +97551.272,E4 +0.000} C_DIS
LIN {X -190.795,Y +1039.355,Z +0.000,A -0.983,E1 +46.842,E3 +97565.932,E4 +0.000} C_DIS
LIN {X -190.395,Y +1028.856,Z +0.000,A -0.089,E1 +46.598,E3 +97579.326,E4 +0.000} C_DIS
LIN {X -190.239,Y +1018.851,Z +0.000,A -0.004,E1 +46.529,E3 +97592.094,E4 +0.000} C_DIS
LIN {X -190.161,Y +1004.975,Z +0.000,A +0.000,E1 +46.506,E3 +97609.808,E4 +0.000} C_DIS
LIN {X -190.142,Y +412.853,Z +0.000,A +0.000,E1 +46.501,E3 +98366.014,E4 +0.000} C_DIS
LIN {X -190.147,Y +401.077,Z +0.000,A +0.000,E1 +46.499,E3 +98381.055,E4 +0.000} C_DIS
LIN {X -190.159,Y +390.929,Z +0.000,A +0.000,E1 +46.494,E3 +98394.021,E4 +0.000} C_DIS
LIN {X -190.174,Y +383.973,Z +0.000,A +0.000,E1 +46.484,E3 +98402.914,E4 +0.000} C_DIS
LIN {X -190.200,Y +373.815,Z +0.000,A +0.000,E1 +46.448,E3 +98415.919,E4 +0.000} C_DIS
LIN {X -190.154,Y +361.003,Z +0.000,A +0.000,E1 +46.303,E3 +98432.413,E4 +0.000} C_DIS
LIN {X -189.772,Y +350.660,Z +0.000,A +0.049,E1 +45.996,E3 +98445.952,E4 +0.000} C_DIS
LIN {X -189.325,Y +346.917,Z +0.000,A +0.243,E1 +45.771,E3 +98451.021,E4 +0.000} C_DIS
LIN {X -188.196,Y +342.754,Z +0.000,A +1.966,E1 +45.249,E3 +98457.029,E4 +0.000} C_DIS
LIN {X -185.199,Y +337.023,Z +0.000,A +6.630,E1 +43.793,E3 +98466.403,E4 +0.000} C_DIS
LIN {X -181.141,Y +331.596,Z +0.000,A +12.274,E1 +41.569,E3 +98476.963,E4 +0.000} C_DIS
LIN {X -176.762,Y +326.804,Z +0.000,A +17.560,E1 +38.898,E3 +98488.387,E4 +0.000} C_DIS
LIN {X -172.184,Y +322.578,Z +0.000,A +19.859,E1 +36.197,E3 +98501.117,E4 +0.000} C_DIS
LIN {X -165.998,Y +317.874,Z +0.000,A +20.000,E1 +32.027,E3 +98520.875,E4 +0.000} C_DIS
LIN {X -160.137,Y +314.334,Z +0.000,A +20.000,E1 +26.368,E3 +98545.244,E4 +0.000} C_DIS
LIN {X -155.624,Y +312.245,Z +0.000,A +20.000,E1 +19.506,E3 +98573.920,E4 +0.000} C_DIS
LIN {X -153.557,Y +311.879,Z +0.000,A +20.000,E1 +11.113,E3 +98609.675,E4 +0.000} C_DIS
LIN {X -155.320,Y +313.348,Z +0.000,A +20.000,E1 +3.401,E3 +98642.859,E4 +0.000} C_DIS
LIN {X -160.005,Y +315.804,Z +0.000,A +20.000,E1 -4.720,E3 +98673.237,E4 +0.000} C_DIS
LIN {X -164.504,Y +318.255,Z +0.000,A +20.000,E1 -10.663,E3 +98692.606,E4 +0.000} C_DIS
LIN {X -170.340,Y +322.684,Z +0.000,A +20.000,E1 -17.457,E3 +98712.638,E4 +0.000} C_DIS
LIN {X -175.568,Y +329.106,Z +0.000,A +20.000,E1 -24.747,E3 +98729.872,E4 +0.000} C_DIS
LIN {X -184.074,Y +340.065,Z +0.000,A +20.000,E1 -33.664,E3 +98752.812,E4 +0.000} C_DIS
LIN {X -190.779,Y +351.388,Z +0.000,A +20.000,E1 -40.083,E3 +98770.590,E4 +0.000} C_DIS
LIN {X -195.254,Y +362.955,Z +0.000,A +20.000,E1 -44.515,E3 +98785.343,E4 +0.000} C_DIS
LIN {X -197.754,Y +374.780,Z +0.000,A +20.000,E1 -47.450,E3 +98798.765,E4 +0.000} C_DIS
LIN {X -198.310,Y +383.215,Z +0.000,A +19.956,E1 -48.698,E3 +98807.889,E4 +0.000} C_DIS
LIN {X -197.912,Y +391.275,Z +0.000,A +18.601,E1 -49.158,E3 +98816.607,E4 +0.000} C_DIS
LIN {X -196.679,Y +398.944,Z +0.000,A +13.989,E1 -48.784,E3 +98825.161,E4 +0.000} C_DIS
LIN {X -194.742,Y +406.288,Z +0.000,A +8.476,E1 -48.001,E3 +98833.844,E4 +0.000} C_DIS
LIN {X -192.748,Y +413.472,Z +0.000,A +3.905,E1 -47.267,E3 +98842.854,E4 +0.000} C_DIS
LIN {X -191.781,Y +419.162,Z +0.000,A +1.739,E1 -46.975,E3 +98850.122,E4 +0.000} C_DIS
LIN {X -190.795,Y +430.646,Z +0.000,A +0.152,E1 -46.707,E3 +98864.783,E4 +0.000} C_DIS
LIN {X -190.395,Y +441.145,Z +0.000,A +0.001,E1 -46.583,E3 +98878.176,E4 +0.000} C_DIS
LIN {X -190.239,Y +451.150,Z +0.000,A -0.000,E1 -46.528,E3 +98890.944,E4 +0.000} C_DIS
LIN {X -190.161,Y +465.026,Z +0.000,A -0.000,E1 -46.506,E3 +98908.659,E4 +0.000} C_DIS
LIN {X -190.142,Y +1057.148,Z +0.000,A -0.000,E1 -46.500,E3 +99664.865,E4 +0.000} C_DIS
LIN {X -190.147,Y +1068.924,Z +0.000,A -0.000,E1 -46.499,E3 +99679.906,E4 +0.000} C_DIS
LIN {X -190.159,Y +1079.072,Z +0.000,A -0.000,E1 -46.493,E3 +99692.871,E4 +0.000} C_DIS
LIN {X -190.174,Y +1086.028,Z +0.000,A -0.000,E1 -46.483,E3 +99701.765,E4 +0.000} C_DIS
LIN {X -190.200,Y +1096.186,Z +0.000,A -0.000,E1 -46.448,E3 +99714.769,E4 +0.000} C_DIS
LIN {X -190.154,Y +1108.998,Z +0.000,A -0.054,E1 -46.295,E3 +99731.264,E4 +0.000} C_DIS
LIN {X -189.772,Y +1119.341,Z +0.000,A -0.752,E1 -45.902,E3 +99744.802,E4 +0.000} C_DIS
LIN {X -189.097,Y +1124.276,Z +0.000,A -2.508,E1 -45.397,E3 +99751.534,E4 +0.000} C_DIS
LIN {X -187.410,Y +1129.069,Z +0.000,A -5.304,E1 -44.585,E3 +99758.707,E4 +0.000} C_DIS
LIN {X -183.899,Y +1134.873,Z +0.000,A -10.372,E1 -42.805,E3 +99768.713,E4 +0.000} C_DIS
LIN {X -179.711,Y +1140.065,Z +0.000,A -15.940,E1 -40.393,E3 +99779.499,E4 +0.000} C_DIS
LIN {X -176.763,Y +1143.197,Z +0.000,A -18.748,E1 -38.674,E3 +99787.237,E4 +0.000} C_DIS
LIN {X -172.185,Y +1147.423,Z +0.000,A -19.971,E1 -36.175,E3 +99799.967,E4 +0.000} C_DIS
LIN {X -165.999,Y +1152.127,Z +0.000,A -20.000,E1 -32.027,E3 +99819.725,E4 +0.000} C_DIS
LIN {X -160.138,Y +1155.667,Z +0.000,A -20.000,E1 -26.368,E3 +99844.095,E4 +0.000} C_DIS
LIN {X -155.625,Y +1157.756,Z +0.000,A -20.000,E1 -19.505,E3 +99872.771,E4 +0.000} C_DIS
LIN {X -153.552,Y +1158.113,Z +0.000,A -20.000,E1 -11.113,E3 +99908.522,E4 +0.000} C_DIS
LIN {X -156.311,Y +1155.540,Z +0.000,A -20.000,E1 -0.839,E3 +99951.882,E4 +0.000} C_DIS
LIN {X -161.281,Y +1151.851,Z +0.000,A -20.000,E1 +7.737,E3 +99981.781,E4 +0.000} C_DIS
LIN {X -167.493,Y +1147.157,Z +0.000,A -20.000,E1 +16.195,E3 +100006.220,E4 +0.000} C_DIS
LIN {X -173.235,Y +1142.221,Z +0.000,A -20.000,E1 +22.930,E3 +100023.522,E4 +0.000} C_DIS
LIN {X -181.123,Y +1133.734,Z +0.000,A -20.000,E1 +30.868,E3 +100044.278,E4 +0.000} C_DIS
LIN {X -189.654,Y +1120.856,Z +0.000,A -20.000,E1 +39.018,E3 +100066.292,E4 +0.000} C_DIS
LIN {X -195.246,Y +1107.046,Z +0.000,A -20.000,E1 +44.515,E3 +100084.194,E4 +0.000} C_DIS
LIN {X -198.051,Y +1092.368,Z +0.000,A -20.000,E1 +47.947,E3 +100100.720,E4 +0.000} C_DIS
LIN {X -198.143,Y +1081.370,Z +0.000,A -19.806,E1 +49.153,E3 +100112.581,E4 +0.000} C_DIS
LIN {X -197.177,Y +1073.569,Z +0.000,A -17.356,E1 +49.162,E3 +100121.165,E4 +0.000} C_DIS
LIN {X -195.448,Y +1066.139,Z +0.000,A -12.154,E1 +48.512,E3 +100129.760,E4 +0.000} C_DIS
LIN {X -193.346,Y +1058.941,Z +0.000,A -7.133,E1 +47.724,E3 +100138.640,E4 +0.000} C_DIS
LIN {X -191.781,Y +1050.839,Z +0.000,A -3.715,E1 +47.274,E3 +100148.973,E4 +0.000} C_DIS
LIN {X -190.795,Y +1039.355,Z +0.000,A -0.983,E1 +46.842,E3 +100163.633,E4 +0.000} C_DIS
LIN {X -190.395,Y +1028.856,Z +0.000,A -0.089,E1 +46.598,E3 +100177.027,E4 +0.000} C_DIS
LIN {X -190.239,Y +1018.851,Z +0.000,A -0.004,E1 +46.529,E3 +100189.795,E4 +0.000} C_DIS
LIN {X -190.161,Y +1004.975,Z +0.000,A +0.000,E1 +46.506,E3 +100207.509,E4 +0.000} C_DIS
LIN {X -190.142,Y +412.853,Z +0.000,A +0.000,E1 +46.501,E3 +100963.715,E4 +0.000} C_DIS
LIN {X -190.147,Y +401.077,Z +0.000,A +0.000,E1 +46.499,E3 +100978.756,E4 +0.000} C_DIS
LIN {X -190.159,Y +390.929,Z +0.000,A +0.000,E1 +46.494,E3 +100991.722,E4 +0.000} C_DIS
LIN {X -190.174,Y +383.973,Z +0.000,A +0.000,E1 +46.484,E3 +101000.615,E4 +0.000} C_DIS
LIN {X -190.200,Y +373.815,Z +0.000,A +0.000,E1 +46.448,E3 +101013.620,E4 +0.000} C_DIS
LIN {X -190.154,Y +361.003,Z +0.000,A +0.000,E1 +46.303,E3 +101030.114,E4 +0.000} C_DIS
LIN {X -189.772,Y +350.660,Z +0.000,A +0.049,E1 +45.996,E3 +101043.653,E4 +0.000} C_DIS
LIN {X -189.325,Y +346.917,Z +0.000,A +0.243,E1 +45.771,E3 +101048.722,E4 +0.000} C_DIS
LIN {X -188.196,Y +342.754,Z +0.000,A +1.966,E1 +45.249,E3 +101054.730,E4 +0.000} C_DIS
LIN {X -185.199,Y +337.023,Z +0.000,A +6.630,E1 +43.793,E3 +101064.104,E4 +0.000} C_DIS
LIN {X -181.141,Y +331.596,Z +0.000,A +12.274,E1 +41.569,E3 +101074.664,E4 +0.000} C_DIS
LIN {X -176.762,Y +326.804,Z +0.000,A +17.560,E1 +38.898,E3 +101086.088,E4 +0.000} C_DIS
LIN {X -172.184,Y +322.578,Z +0.000,A +19.859,E1 +36.197,E3 +101098.818,E4 +0.000} C_DIS
LIN {X -165.998,Y +317.874,Z +0.000,A +20.000,E1 +32.027,E3 +101118.576,E4 +0.000} C_DIS
LIN {X -160.137,Y +314.334,Z +0.000,A +20.000,E1 +26.368,E3 +101142.945,E4 +0.000} C_DIS
LIN {X -155.624,Y +312.245,Z +0.000,A +20.000,E1 +19.506,E3 +101171.621,E4 +0.000} C_DIS
LIN {X -153.557,Y +311.879,Z +0.000,A +20.000,E1 +11.113,E3 +101207.376,E4 +0.000} C_DIS
LIN {X -155.320,Y +313.348,Z +0.000,A +20.000,E1 +3.401,E3 +101240.560,E4 +0.000} C_DIS
LIN {X -160.005,Y +315.804,Z +0.000,A +20.000,E1 -4.720,E3 +101270.938,E4 +0.000} C_DIS
LIN {X -164.504,Y +318.255,Z +0.000,A +20.000,E1 -10.663,E3 +101290.307,E4 +0.000} C_DIS
LIN {X -170.340,Y +322.684,Z +0.000,A +20.000,E1 -17.457,E3 +101310.339,E4 +0.000} C_DIS
LIN {X -175.568,Y +329.106,Z +0.000,A +20.000,E1 -24.747,E3 +101327.573,E4 +0.000} C_DIS
LIN {X -184.074,Y +340.065,Z +0.000,A +20.000,E1 -33.664,E3 +101350.513,E4 +0.000} C_DIS
LIN {X -190.779,Y +351.388,Z +0.000,A +20.000,E1 -40.083,E3 +101368.291,E4 +0.000} C_DIS
LIN {X -195.254,Y +362.955,Z +0.000,A +20.000,E1 -44.515,E3 +101383.044,E4 +0.000} C_DIS
LIN {X -197.754,Y +374.780,Z +0.000,A +20.000,E1 -47.450,E3 +101396.466,E4 +0.000} C_DIS
LIN {X -198.310,Y +383.215,Z +0.000,A +19.956,E1 -48.698,E3 +101405.590,E4 +0.000} C_DIS
LIN {X -197.912,Y +391.275,Z +0.000,A +18.601,E1 -49.158,E3 +101414.308,E4 +0.000} C_DIS
LIN {X -196.679,Y +398.944,Z +0.000,A +13.989,E1 -48.784,E3 +101422.862,E4 +0.000} C_DIS
LIN {X -194.742,Y +406.288,Z +0.000,A +8.476,E1 -48.001,E3 +101431.545,E4 +0.000} C_DIS
LIN {X -192.748,Y +413.472,Z +0.000,A +3.905,E1 -47.267,E3 +101440.555,E4 +0.000} C_DIS
LIN {X -191.781,Y +419.162,Z +0.000,A +1.739,E1 -46.975,E3 +101447.823,E4 +0.000} C_DIS
LIN {X -190.795,Y +430.646,Z +0.000,A +0.152,E1 -46.707,E3 +101462.484,E4 +0.000} C_DIS
LIN {X -190.395,Y +441.145,Z +0.000,A +0.001,E1 -46.583,E3 +101475.877,E4 +0.000} C_DIS
LIN {X -190.239,Y +451.150,Z +0.000,A -0.000,E1 -46.528,E3 +101488.645,E4 +0.000} C_DIS
LIN {X -190.161,Y +465.026,Z +0.000,A -0.000,E1 -46.506,E3 +101506.360,E4 +0.000} C_DIS
LIN {X -190.142,Y +1057.148,Z +0.000,A -0.000,E1 -46.500,E3 +102262.566,E4 +0.000} C_DIS
LIN {X -190.147,Y +1068.924,Z +0.000,A -0.000,E1 -46.499,E3 +102277.607,E4 +0.000} C_DIS
LIN {X -190.159,Y +1079.072,Z +0.000,A -0.000,E1 -46.493,E3 +102290.572,E4 +0.000} C_DIS
LIN {X -190.174,Y +1086.028,Z +0.000,A -0.000,E1 -46.483,E3 +102299.466,E4 +0.000} C_DIS
LIN {X -190.200,Y +1096.186,Z +0.000,A -0.000,E1 -46.448,E3 +102312.470,E4 +0.000} C_DIS
LIN {X -190.154,Y +1108.998,Z +0.000,A -0.054,E1 -46.295,E3 +102328.965,E4 +0.000} C_DIS
LIN {X -189.772,Y +1119.341,Z +0.000,A -0.752,E1 -45.902,E3 +102342.503,E4 +0.000} C_DIS
LIN {X -189.097,Y +1124.276,Z +0.000,A -2.508,E1 -45.397,E3 +102349.235,E4 +0.000} C_DIS
LIN {X -187.410,Y +1129.069,Z +0.000,A -5.304,E1 -44.585,E3 +102356.408,E4 +0.000} C_DIS
LIN {X -183.899,Y +1134.873,Z +0.000,A -10.372,E1 -42.805,E3 +102366.414,E4 +0.000} C_DIS
LIN {X -179.711,Y +1140.065,Z +0.000,A -15.940,E1 -40.393,E3 +102377.200,E4 +0.000} C_DIS
LIN {X -176.763,Y +1143.197,Z +0.000,A -18.748,E1 -38.674,E3 +102384.938,E4 +0.000} C_DIS
LIN {X -172.185,Y +1147.423,Z +0.000,A -19.971,E1 -36.175,E3 +102397.668,E4 +0.000} C_DIS
LIN {X -165.999,Y +1152.127,Z +0.000,A -20.000,E1 -32.027,E3 +102417.426,E4 +0.000} C_DIS
LIN {X -160.138,Y +1155.667,Z +0.000,A -20.000,E1 -26.368,E3 +102441.796,E4 +0.000} C_DIS
LIN {X -155.625,Y +1157.756,Z +0.000,A -20.000,E1 -19.505,E3 +102470.472,E4 +0.000} C_DIS
LIN {X -153.552,Y +1158.113,Z +0.000,A -20.000,E1 -11.113,E3 +102506.223,E4 +0.000} C_DIS
LIN {X -156.311,Y +1155.540,Z +0.000,A -20.000,E1 -0.839,E3 +102549.583,E4 +0.000} C_DIS
LIN {X -161.281,Y +1151.851,Z +0.000,A -20.000,E1 +7.737,E3 +102579.482,E4 +0.000} C_DIS
LIN {X -167.493,Y +1147.157,Z +0.000,A -20.000,E1 +16.195,E3 +102603.921,E4 +0.000} C_DIS
LIN {X -173.235,Y +1142.221,Z +0.000,A -20.000,E1 +22.930,E3 +102621.223,E4 +0.000} C_DIS
LIN {X -181.123,Y +1133.734,Z +0.000,A -20.000,E1 +30.868,E3 +102641.979,E4 +0.000} C_DIS
LIN {X -189.654,Y +1120.856,Z +0.000,A -20.000,E1 +39.018,E3 +102663.993,E4 +0.000} C_DIS
LIN {X -195.246,Y +1107.046,Z +0.000,A -20.000,E1 +44.515,E3 +102681.895,E4 +0.000} C_DIS
LIN {X -198.051,Y +1092.368,Z +0.000,A -20.000,E1 +47.947,E3 +102698.421,E4 +0.000} C_DIS
LIN {X -198.143,Y +1081.370,Z +0.000,A -19.806,E1 +49.153,E3 +102710.282,E4 +0.000} C_DIS
LIN {X -197.177,Y +1073.569,Z +0.000,A -17.356,E1 +49.162,E3 +102718.866,E4 +0.000} C_DIS
LIN {X -195.448,Y +1066.139,Z +0.000,A -12.154,E1 +48.512,E3 +102727.461,E4 +0.000} C_DIS
LIN {X -193.346,Y +1058.941,Z +0.000,A -7.133,E1 +47.724,E3 +102736.341,E4 +0.000} C_DIS
LIN {X -191.781,Y +1050.839,Z +0.000,A -3.715,E1 +47.274,E3 +102746.674,E4 +0.000} C_DIS
LIN {X -190.795,Y +1039.355,Z +0.000,A -0.983,E1 +46.842,E3 +102761.334,E4 +0.000} C_DIS
LIN {X -190.395,Y +1028.856,Z +0.000,A -0.089,E1 +46.598,E3 +102774.728,E4 +0.000} C_DIS
LIN {X -190.239,Y +1018.851,Z +0.000,A -0.004,E1 +46.529,E3 +102787.496,E4 +0.000} C_DIS
LIN {X -190.161,Y +1004.975,Z +0.000,A +0.000,E1 +46.506,E3 +102805.210,E4 +0.000} C_DIS
LIN {X -190.142,Y +412.853,Z +0.000,A +0.000,E1 +46.501,E3 +103561.416,E4 +0.000} C_DIS
LIN {X -190.147,Y +401.077,Z +0.000,A +0.000,E1 +46.499,E3 +103576.457,E4 +0.000} C_DIS
LIN {X -190.159,Y +390.929,Z +0.000,A +0.000,E1 +46.494,E3 +103589.423,E4 +0.000} C_DIS
LIN {X -190.174,Y +383.973,Z +0.000,A +0.000,E1 +46.484,E3 +103598.316,E4 +0.000} C_DIS
LIN {X -190.200,Y +373.815,Z +0.000,A +0.000,E1 +46.448,E3 +103611.321,E4 +0.000} C_DIS
LIN {X -190.154,Y +361.003,Z +0.000,A +0.000,E1 +46.303,E3 +103627.815,E4 +0.000} C_DIS
LIN {X -189.772,Y +350.660,Z +0.000,A +0.049,E1 +45.996,E3 +103641.354,E4 +0.000} C_DIS
LIN {X -189.325,Y +346.917,Z +0.000,A +0.243,E1 +45.771,E3 +103646.423,E4 +0.000} C_DIS
LIN {X -188.196,Y +342.754,Z +0.000,A +1.966,E1 +45.249,E3 +103652.431,E4 +0.000} C_DIS
LIN {X -185.199,Y +337.023,Z +0.000,A +6.630,E1 +43.793,E3 +103661.805,E4 +0.000} C_DIS
LIN {X -181.141,Y +331.596,Z +0.000,A +12.274,E1 +41.569,E3 +103672.365,E4 +0.000} C_DIS
LIN {X -176.762,Y +326.804,Z +0.000,A +17.560,E1 +38.898,E3 +103683.789,E4 +0.000} C_DIS
LIN {X -172.184,Y +322.578,Z +0.000,A +19.859,E1 +36.197,E3 +103696.519,E4 +0.000} C_DIS
LIN {X -165.998,Y +317.874,Z +0.000,A +20.000,E1 +32.027,E3 +103716.277,E4 +0.000} C_DIS
LIN {X -160.137,Y +314.334,Z +0.000,A +20.000,E1 +26.368,E3 +103740.646,E4 +0.000} C_DIS
LIN {X -155.624,Y +312.245,Z +0.000,A +20.000,E1 +19.506,E3 +103769.322,E4 +0.000} C_DIS
LIN {X -153.557,Y +311.879,Z +0.000,A +20.000,E1 +11.113,E3 +103805.077,E4 +0.000} C_DIS
LIN {X -155.320,Y +313.348,Z +0.000,A +20.000,E1 +3.401,E3 +103838.261,E4 +0.000} C_DIS
LIN {X -160.005,Y +315.804,Z +0.000,A +20.000,E1 -4.720,E3 +103868.639,E4 +0.000} C_DIS
LIN {X -164.504,Y +318.255,Z +0.000,A +20.000,E1 -10.663,E3 +103888.008,E4 +0.000} C_DIS
LIN {X -170.340,Y +322.684,Z +0.000,A +20.000,E1 -17.457,E3 +103908.040,E4 +0.000} C_DIS
LIN {X -175.568,Y +329.106,Z +0.000,A +20.000,E1 -24.747,E3 +103925.274,E4 +0.000} C_DIS
LIN {X -184.074,Y +340.065,Z +0.000,A +20.000,E1 -33.664,E3 +103948.214,E4 +0.000} C_DIS
LIN {X -190.779,Y +351.388,Z +0.000,A +20.000,E1 -40.083,E3 +103965.992,E4 +0.000} C_DIS
LIN {X -195.254,Y +362.955,Z +0.000,A +20.000,E1 -44.515,E3 +103980.745,E4 +0.000} C_DIS
LIN {X -197.754,Y +374.780,Z +0.000,A +20.000,E1 -47.450,E3 +103994.167,E4 +0.000} C_DIS
LIN {X -198.310,Y +383.215,Z +0.000,A +19.956,E1 -48.698,E3 +104003.291,E4 +0.000} C_DIS
LIN {X -197.912,Y +391.275,Z +0.000,A +18.601,E1 -49.158,E3 +104012.009,E4 +0.000} C_DIS
LIN {X -196.679,Y +398.944,Z +0.000,A +13.989,E1 -48.784,E3 +104020.563,E4 +0.000} C_DIS
LIN {X -194.742,Y +406.288,Z +0.000,A +8.476,E1 -48.001,E3 +104029.246,E4 +0.000} C_DIS
LIN {X -192.748,Y +413.472,Z +0.000,A +3.905,E1 -47.267,E3 +104038.256,E4 +0.000} C_DIS
LIN {X -191.781,Y +419.162,Z +0.000,A +1.739,E1 -46.975,E3 +104045.524,E4 +0.000} C_DIS
LIN {X -190.795,Y +430.646,Z +0.000,A +0.152,E1 -46.707,E3 +104060.185,E4 +0.000} C_DIS
LIN {X -190.395,Y +441.145,Z +0.000,A +0.001,E1 -46.583,E3 +104073.578,E4 +0.000} C_DIS
LIN {X -190.239,Y +451.150,Z +0.000,A -0.000,E1 -46.528,E3 +104086.346,E4 +0.000} C_DIS
LIN {X -190.161,Y +465.026,Z +0.000,A -0.000,E1 -46.506,E3 +104104.061,E4 +0.000} C_DIS
LIN {X -190.142,Y +1057.148,Z +0.000,A -0.000,E1 -46.500,E3 +104860.267,E4 +0.000} C_DIS
LIN {X -190.147,Y +1068.924,Z +0.000,A -0.000,E1 -46.499,E3 +104875.308,E4 +0.000} C_DIS
LIN {X -190.159,Y +1079.072,Z +0.000,A -0.000,E1 -46.493,E3 +104888.273,E4 +0.000} C_DIS
LIN {X -190.174,Y +1086.028,Z +0.000,A -0.000,E1 -46.483,E3 +104897.167,E4 +0.000} C_DIS
LIN {X -190.200,Y +1096.186,Z +0.000,A -0.000,E1 -46.448,E3 +104910.171,E4 +0.000} C_DIS
LIN {X -190.154,Y +1108.998,Z +0.000,A -0.054,E1 -46.295,E3 +104926.666,E4 +0.000} C_DIS
LIN {X -189.772,Y +1119.341,Z +0.000,A -0.752,E1 -45.902,E3 +104940.204,E4 +0.000} C_DIS
LIN {X -189.097,Y +1124.276,Z +0.000,A -2.508,E1 -45.397,E3 +104946.936,E4 +0.000} C_DIS
LIN {X -187.410,Y +1129.069,Z +0.000,A -5.304,E1 -44.585,E3 +104954.109,E4 +0.000} C_DIS
LIN {X -183.899,Y +1134.873,Z +0.000,A -10.372,E1 -42.805,E3 +104964.115,E4 +0.000} C_DIS
LIN {X -179.711,Y +1140.065,Z +0.000,A -15.940,E1 -40.393,E3 +104974.901,E4 +0.000} C_DIS
LIN {X -176.763,Y +1143.197,Z +0.000,A -18.748,E1 -38.674,E3 +104982.639,E4 +0.000} C_DIS
LIN {X -172.185,Y +1147.423,Z +0.000,A -19.971,E1 -36.175,E3 +104995.369,E4 +0.000} C_DIS
LIN {X -165.999,Y +1152.127,Z +0.000,A -20.000,E1 -32.027,E3 +105015.127,E4 +0.000} C_DIS
LIN {X -160.138,Y +1155.667,Z +0.000,A -20.000,E1 -26.368,E3 +105039.497,E4 +0.000} C_DIS
LIN {X -155.625,Y +1157.756,Z +0.000,A -20.000,E1 -19.505,E3 +105068.173,E4 +0.000} C_DIS
LIN {X -153.552,Y +1158.113,Z +0.000,A -20.000,E1 -11.113,E3 +105103.924,E4 +0.000} C_DIS
LIN {X -156.311,Y +1155.540,Z +0.000,A -20.000,E1 -0.839,E3 +105147.284,E4 +0.000} C_DIS
LIN {X -161.281,Y +1151.851,Z +0.000,A -20.000,E1 +7.737,E3 +105177.183,E4 +0.000} C_DIS
LIN {X -167.493,Y +1147.157,Z +0.000,A -20.000,E1 +16.195,E3 +105201.622,E4 +0.000} C_DIS
LIN {X -173.235,Y +1142.221,Z +0.000,A -20.000,E1 +22.930,E3 +105218.924,E4 +0.000} C_DIS
LIN {X -181.123,Y +1133.734,Z +0.000,A -20.000,E1 +30.868,E3 +105239.680,E4 +0.000} C_DIS
LIN {X -189.654,Y +1120.856,Z +0.000,A -20.000,E1 +39.018,E3 +105261.694,E4 +0.000} C_DIS
LIN {X -195.246,Y +1107.046,Z +0.000,A -20.000,E1 +44.515,E3 +105279.596,E4 +0.000} C_DIS
LIN {X -198.051,Y +1092.368,Z +0.000,A -20.000,E1 +47.947,E3 +105296.122,E4 +0.000} C_DIS
LIN {X -198.143,Y +1081.370,Z +0.000,A -19.806,E1 +49.153,E3 +105307.983,E4 +0.000} C_DIS
LIN {X -197.177,Y +1073.569,Z +0.000,A -17.356,E1 +49.162,E3 +105316.567,E4 +0.000} C_DIS
LIN {X -195.448,Y +1066.139,Z +0.000,A -12.154,E1 +48.512,E3 +105325.162,E4 +0.000} C_DIS
LIN {X -193.346,Y +1058.941,Z +0.000,A -7.133,E1 +47.724,E3 +105334.042,E4 +0.000} C_DIS
LIN {X -191.781,Y +1050.839,Z +0.000,A -3.715,E1 +47.274,E3 +105344.375,E4 +0.000} C_DIS
LIN {X -190.795,Y +1039.355,Z +0.000,A -0.983,E1 +46.842,E3 +105359.035,E4 +0.000} C_DIS
LIN {X -190.395,Y +1028.856,Z +0.000,A -0.089,E1 +46.598,E3 +105372.429,E4 +0.000} C_DIS
LIN {X -190.239,Y +1018.851,Z +0.000,A -0.004,E1 +46.529,E3 +105385.197,E4 +0.000} C_DIS
LIN {X -190.161,Y +1004.975,Z +0.000,A +0.000,E1 +46.506,E3 +105402.911,E4 +0.000} C_DIS
LIN {X -190.142,Y +412.853,Z +0.000,A +0.000,E1 +46.501,E3 +106159.117,E4 +0.000} C_DIS
LIN {X -190.147,Y +401.077,Z +0.000,A +0.000,E1 +46.499,E3 +106174.158,E4 +0.000} C_DIS
LIN {X -190.159,Y +390.929,Z +0.000,A +0.000,E1 +46.494,E3 +106187.124,E4 +0.000} C_DIS
LIN {X -190.174,Y +383.973,Z +0.000,A +0.000,E1 +46.484,E3 +106196.017,E4 +0.000} C_DIS
LIN {X -190.200,Y +373.815,Z +0.000,A +0.000,E1 +46.448,E3 +106209.022,E4 +0.000} C_DIS
LIN {X -190.154,Y +361.003,Z +0.000,A +0.000,E1 +46.303,E3 +106225.516,E4 +0.000} C_DIS
LIN {X -189.772,Y +350.660,Z +0.000,A +0.049,E1 +45.996,E3 +106239.055,E4 +0.000} C_DIS
LIN {X -189.325,Y +346.917,Z +0.000,A +0.243,E1 +45.771,E3 +106244.124,E4 +0.000} C_DIS
LIN {X -188.196,Y +342.754,Z +0.000,A +1.966,E1 +45.249,E3 +106250.132,E4 +0.000} C_DIS
LIN {X -185.199,Y +337.023,Z +0.000,A +6.630,E1 +43.793,E3 +106259.506,E4 +0.000} C_DIS
LIN {X -181.141,Y +331.596,Z +0.000,A +12.274,E1 +41.569,E3 +106270.066,E4 +0.000} C_DIS
LIN {X -176.762,Y +326.804,Z +0.000,A +17.560,E1 +38.898,E3 +106281.490,E4 +0.000} C_DIS
LIN {X -172.184,Y +322.578,Z +0.000,A +19.859,E1 +36.197,E3 +106294.220,E4 +0.000} C_DIS
LIN {X -165.998,Y +317.874,Z +0.000,A +20.000,E1 +32.027,E3 +106313.978,E4 +0.000} C_DIS
LIN {X -160.137,Y +314.334,Z +0.000,A +20.000,E1 +26.368,E3 +106338.347,E4 +0.000} C_DIS
LIN {X -155.624,Y +312.245,Z +0.000,A +20.000,E1 +19.506,E3 +106367.023,E4 +0.000} C_DIS
LIN {X -153.557,Y +311.879,Z +0.000,A +20.000,E1 +11.113,E3 +106402.778,E4 +0.000} C_DIS
LIN {X -155.320,Y +313.348,Z +0.000,A +20.000,E1 +3.401,E3 +106435.962,E4 +0.000} C_DIS
LIN {X -160.005,Y +315.804,Z +0.000,A +20.000,E1 -4.720,E3 +106466.340,E4 +0.000} C_DIS
LIN {X -164.504,Y +318.255,Z +0.000,A +20.000,E1 -10.663,E3 +106485.709,E4 +0.000} C_DIS
LIN {X -170.340,Y +322.684,Z +0.000,A +20.000,E1 -17.457,E3 +106505.741,E4 +0.000} C_DIS
LIN {X -175.568,Y +329.106,Z +0.000,A +20.000,E1 -24.747,E3 +106522.975,E4 +0.000} C_DIS
LIN {X -184.074,Y +340.065,Z +0.000,A +20.000,E1 -33.664,E3 +106545.915,E4 +0.000} C_DIS
LIN {X -190.779,Y +351.388,Z +0.000,A +20.000,E1 -40.083,E3 +106563.693,E4 +0.000} C_DIS
LIN {X -195.254,Y +362.955,Z +0.000,A +20.000,E1 -44.515,E3 +106578.446,E4 +0.000} C_DIS
LIN {X -197.754,Y +374.780,Z +0.000,A +20.000,E1 -47.450,E3 +106591.868,E4 +0.000} C_DIS
LIN {X -198.310,Y +383.215,Z +0.000,A +19.956,E1 -48.698,E3 +106600.992,E4 +0.000} C_DIS
LIN {X -197.912,Y +391.275,Z +0.000,A +18.601,E1 -49.158,E3 +106609.710,E4 +0.000} C_DIS
LIN {X -196.679,Y +398.944,Z +0.000,A +13.989,E1 -48.784,E3 +106618.264,E4 +0.000} C_DIS
LIN {X -194.742,Y +406.288,Z +0.000,A +8.476,E1 -48.001,E3 +106626.947,E4 +0.000} C_DIS
LIN {X -192.748,Y +413.472,Z +0.000,A +3.905,E1 -47.267,E3 +106635.957,E4 +0.000} C_DIS
LIN {X -191.781,Y +419.162,Z +0.000,A +1.739,E1 -46.975,E3 +106643.225,E4 +0.000} C_DIS
LIN {X -190.795,Y +430.646,Z +0.000,A +0.152,E1 -46.707,E3 +106657.886,E4 +0.000} C_DIS
LIN {X -190.395,Y +441.145,Z +0.000,A +0.001,E1 -46.583,E3 +106671.279,E4 +0.000} C_DIS
LIN {X -190.239,Y +451.150,Z +0.000,A -0.000,E1 -46.528,E3 +106684.047,E4 +0.000} C_DIS
LIN {X -190.161,Y +465.026,Z +0.000,A -0.000,E1 -46.506,E3 +106701.762,E4 +0.000} C_DIS
LIN {X -190.142,Y +1057.148,Z +0.000,A -0.000,E1 -46.500,E3 +107457.968,E4 +0.000} C_DIS
LIN {X -190.147,Y +1068.924,Z +0.000,A -0.000,E1 -46.499,E3 +107473.009,E4 +0.000} C_DIS
LIN {X -190.159,Y +1079.072,Z +0.000,A -0.000,E1 -46.493,E3 +107485.974,E4 +0.000} C_DIS
LIN {X -190.174,Y +1086.028,Z +0.000,A -0.000,E1 -46.483,E3 +107494.868,E4 +0.000} C_DIS
LIN {X -190.200,Y +1096.186,Z +0.000,A -0.000,E1 -46.448,E3 +107507.872,E4 +0.000} C_DIS
LIN {X -190.154,Y +1108.998,Z +0.000,A -0.054,E1 -46.295,E3 +107524.367,E4 +0.000} C_DIS
LIN {X -189.772,Y +1119.341,Z +0.000,A -0.752,E1 -45.902,E3 +107537.905,E4 +0.000} C_DIS
LIN {X -189.097,Y +1124.276,Z +0.000,A -2.508,E1 -45.397,E3 +107544.637,E4 +0.000} C_DIS
LIN {X -187.410,Y +1129.069,Z +0.000,A -5.304,E1 -44.585,E3 +107551.810,E4 +0.000} C_DIS
LIN {X -183.899,Y +1134.873,Z +0.000,A -10.372,E1 -42.805,E3 +107561.816,E4 +0.000} C_DIS
LIN {X -179.711,Y +1140.065,Z +0.000,A -15.940,E1 -40.393,E3 +107572.602,E4 +0.000} C_DIS
LIN {X -176.763,Y +1143.197,Z +0.000,A -18.748,E1 -38.674,E3 +107580.340,E4 +0.000} C_DIS
LIN {X -172.185,Y +1147.423,Z +0.000,A -19.971,E1 -36.175,E3 +107593.070,E4 +0.000} C_DIS
LIN {X -165.999,Y +1152.127,Z +0.000,A -20.000,E1 -32.027,E3 +107612.828,E4 +0.000} C_DIS
LIN {X -160.138,Y +1155.667,Z +0.000,A -20.000,E1 -26.368,E3 +107637.198,E4 +0.000} C_DIS
LIN {X -155.625,Y +1157.756,Z +0.000,A -20.000,E1 -19.505,E3 +107665.874,E4 +0.000} C_DIS
LIN {X -153.552,Y +1158.113,Z +0.000,A -20.000,E1 -11.113,E3 +107701.625,E4 +0.000} C_DIS
LIN {X -156.311,Y +1155.540,Z +0.000,A -20.000,E1 -0.839,E3 +107744.985,E4 +0.000} C_DIS
LIN {X -161.281,Y +1151.851,Z +0.000,A -20.000,E1 +7.737,E3 +107774.884,E4 +0.000} C_DIS
LIN {X -167.493,Y +1147.157,Z +0.000,A -20.000,E1 +16.195,E3 +107799.323,E4 +0.000} C_DIS
LIN {X -173.235,Y +1142.221,Z +0.000,A -20.000,E1 +22.930,E3 +107816.625,E4 +0.000} C_DIS
LIN {X -181.123,Y +1133.734,Z +0.000,A -20.000,E1 +30.868,E3 +107837.381,E4 +0.000} C_DIS
LIN {X -189.654,Y +1120.856,Z +0.000,A -20.000,E1 +39.018,E3 +107859.395,E4 +0.000} C_DIS
LIN {X -195.246,Y +1107.046,Z +0.000,A -20.000,E1 +44.515,E3 +107877.297,E4 +0.000} C_DIS
LIN {X -198.051,Y +1092.368,Z +0.000,A -20.000,E1 +47.947,E3 +107893.823,E4 +0.000} C_DIS
LIN {X -198.143,Y +1081.370,Z +0.000,A -19.806,E1 +49.153,E3 +107905.684,E4 +0.000} C_DIS
LIN {X -197.177,Y +1073.569,Z +0.000,A -17.356,E1 +49.162,E3 +107914.268,E4 +0.000} C_DIS
LIN {X -195.448,Y +1066.139,Z +0.000,A -12.154,E1 +48.512,E3 +107922.863,E4 +0.000} C_DIS
LIN {X -193.346,Y +1058.941,Z +0.000,A -7.133,E1 +47.724,E3 +107931.743,E4 +0.000} C_DIS
LIN {X -191.781,Y +1050.839,Z +0.000,A -3.715,E1 +47.274,E3 +107942.076,E4 +0.000} C_DIS
LIN {X -190.795,Y +1039.355,Z +0.000,A -0.983,E1 +46.842,E3 +107956.736,E4 +0.000} C_DIS
LIN {X -190.395,Y +1028.856,Z +0.000,A -0.089,E1 +46.598,E3 +107970.130,E4 +0.000} C_DIS
LIN {X -190.239,Y +1018.851,Z +0.000,A -0.004,E1 +46.529,E3 +107982.898,E4 +0.000} C_DIS
LIN {X -190.161,Y +1004.975,Z +0.000,A +0.000,E1 +46.506,E3 +108000.612,E4 +0.000} C_DIS
LIN {X -190.142,Y +412.853,Z +0.000,A +0.000,E1 +46.501,E3 +108756.818,E4 +0.000} C_DIS
LIN {X -190.147,Y +401.077,Z +0.000,A +0.000,E1 +46.499,E3 +108771.859,E4 +0.000} C_DIS
LIN {X -190.159,Y +390.929,Z +0.000,A +0.000,E1 +46.494,E3 +108784.825,E4 +0.000} C_DIS
LIN {X -190.174,Y +383.973,Z +0.000,A +0.000,E1 +46.484,E3 +108793.718,E4 +0.000} C_DIS
LIN {X -190.200,Y +373.815,Z +0.000,A +0.000,E1 +46.448,E3 +108806.723,E4 +0.000} C_DIS
LIN {X -190.154,Y +361.003,Z +0.000,A +0.000,E1 +46.303,E3 +108823.217,E4 +0.000} C_DIS
LIN {X -189.772,Y +350.660,Z +0.000,A +0.049,E1 +45.996,E3 +108836.756,E4 +0.000} C_DIS
LIN {X -189.325,Y +346.917,Z +0.000,A +0.243,E1 +45.771,E3 +108841.825,E4 +0.000} C_DIS
LIN {X -188.196,Y +342.754,Z +0.000,A +1.966,E1 +45.249,E3 +108847.833,E4 +0.000} C_DIS
LIN {X -185.199,Y +337.023,Z +0.000,A +6.630,E1 +43.793,E3 +108857.207,E4 +0.000} C_DIS
LIN {X -181.141,Y +331.596,Z +0.000,A +12.274,E1 +41.569,E3 +108867.767,E4 +0.000} C_DIS
LIN {X -176.762,Y +326.804,Z +0.000,A +17.560,E1 +38.898,E3 +108879.191,E4 +0.000} C_DIS
LIN {X -172.184,Y +322.578,Z +0.000,A +19.859,E1 +36.197,E3 +108891.921,E4 +0.000} C_DIS
LIN {X -165.998,Y +317.874,Z +0.000,A +20.000,E1 +32.027,E3 +108911.679,E4 +0.000} C_DIS
LIN {X -160.137,Y +314.334,Z +0.000,A +20.000,E1 +26.368,E3 +108936.048,E4 +0.000} C_DIS
LIN {X -155.624,Y +312.245,Z +0.000,A +20.000,E1 +19.506,E3 +108964.724,E4 +0.000} C_DIS
LIN {X -153.557,Y +311.879,Z +0.000,A +20.000,E1 +11.113,E3 +109000.479,E4 +0.000} C_DIS
LIN {X -155.320,Y +313.348,Z +0.000,A +20.000,E1 +3.401,E3 +109033.663,E4 +0.000} C_DIS
LIN {X -160.005,Y +315.804,Z +0.000,A +20.000,E1 -4.720,E3 +109064.041,E4 +0.000} C_DIS
LIN {X -164.504,Y +318.255,Z +0.000,A +20.000,E1 -10.663,E3 +109083.410,E4 +0.000} C_DIS
LIN {X -170.340,Y +322.684,Z +0.000,A +20.000,E1 -17.457,E3 +109103.442,E4 +0.000} C_DIS
LIN {X -175.568,Y +329.106,Z +0.000,A +20.000,E1 -24.747,E3 +109120.676,E4 +0.000} C_DIS
LIN {X -184.074,Y +340.065,Z +0.000,A +20.000,E1 -33.664,E3 +109143.616,E4 +0.000} C_DIS
LIN {X -190.779,Y +351.388,Z +0.000,A +20.000,E1 -40.083,E3 +109161.394,E4 +0.000} C_DIS
LIN {X -195.254,Y +362.955,Z +0.000,A +20.000,E1 -44.515,E3 +109176.147,E4 +0.000} C_DIS
LIN {X -197.754,Y +374.780,Z +0.000,A +20.000,E1 -47.450,E3 +109189.569,E4 +0.000} C_DIS
LIN {X -198.310,Y +383.215,Z +0.000,A +19.956,E1 -48.698,E3 +109198.693,E4 +0.000} C_DIS
LIN {X -197.912,Y +391.275,Z +0.000,A +18.601,E1 -49.158,E3 +109207.411,E4 +0.000} C_DIS
LIN {X -196.679,Y +398.944,Z +0.000,A +13.989,E1 -48.784,E3 +109215.965,E4 +0.000} C_DIS
LIN {X -194.742,Y +406.288,Z +0.000,A +8.476,E1 -48.001,E3 +109224.648,E4 +0.000} C_DIS
LIN {X -192.748,Y +413.472,Z +0.000,A +3.905,E1 -47.267,E3 +109233.658,E4 +0.000} C_DIS
LIN {X -191.781,Y +419.162,Z +0.000,A +1.739,E1 -46.975,E3 +109240.926,E4 +0.000} C_DIS
LIN {X -190.795,Y +430.646,Z +0.000,A +0.152,E1 -46.707,E3 +109255.587,E4 +0.000} C_DIS
LIN {X -190.395,Y +441.145,Z +0.000,A +0.001,E1 -46.583,E3 +109268.980,E4 +0.000} C_DIS
LIN {X -190.239,Y +451.150,Z +0.000,A -0.000,E1 -46.528,E3 +109281.748,E4 +0.000} C_DIS
LIN {X -190.161,Y +465.026,Z +0.000,A -0.000,E1 -46.506,E3 +109299.463,E4 +0.000} C_DIS
LIN {X -190.142,Y +1057.148,Z +0.000,A -0.000,E1 -46.500,E3 +110055.669,E4 +0.000} C_DIS
LIN {X -190.147,Y +1068.924,Z +0.000,A -0.000,E1 -46.499,E3 +110070.710,E4 +0.000} C_DIS
LIN {X -190.159,Y +1079.072,Z +0.000,A -0.000,E1 -46.493,E3 +110083.675,E4 +0.000} C_DIS
LIN {X -190.174,Y +1086.028,Z +0.000,A -0.000,E1 -46.483,E3 +110092.569,E4 +0.000} C_DIS
LIN {X -190.200,Y +1096.186,Z +0.000,A -0.000,E1 -46.448,E3 +110105.573,E4 +0.000} C_DIS
LIN {X -190.154,Y +1108.998,Z +0.000,A -0.054,E1 -46.295,E3 +110122.068,E4 +0.000} C_DIS
LIN {X -189.772,Y +1119.341,Z +0.000,A -0.752,E1 -45.902,E3 +110135.606,E4 +0.000} C_DIS
LIN {X -189.097,Y +1124.276,Z +0.000,A -2.508,E1 -45.397,E3 +110142.338,E4 +0.000} C_DIS
LIN {X -187.410,Y +1129.069,Z +0.000,A -5.304,E1 -44.585,E3 +110149.511,E4 +0.000} C_DIS
LIN {X -183.899,Y +1134.873,Z +0.000,A -10.372,E1 -42.805,E3 +110159.517,E4 +0.000} C_DIS
LIN {X -179.711,Y +1140.065,Z +0.000,A -15.940,E1 -40.393,E3 +110170.303,E4 +0.000} C_DIS
LIN {X -176.763,Y +1143.197,Z +0.000,A -18.748,E1 -38.674,E3 +110178.041,E4 +0.000} C_DIS
LIN {X -172.185,Y +1147.423,Z +0.000,A -19.971,E1 -36.175,E3 +110190.771,E4 +0.000} C_DIS
LIN {X -165.999,Y +1152.127,Z +0.000,A -20.000,E1 -32.027,E3 +110210.529,E4 +0.000} C_DIS
LIN {X -160.138,Y +1155.667,Z +0.000,A -20.000,E1 -26.368,E3 +110234.899,E4 +0.000} C_DIS
LIN {X -155.625,Y +1157.756,Z +0.000,A -20.000,E1 -19.505,E3 +110263.575,E4 +0.000} C_DIS
LIN {X -153.552,Y +1158.113,Z +0.000,A -20.000,E1 -11.113,E3 +110299.326,E4 +0.000} C_DIS
LIN {X -156.311,Y +1155.540,Z +0.000,A -20.000,E1 -0.839,E3 +110342.686,E4 +0.000} C_DIS
LIN {X -161.281,Y +1151.851,Z +0.000,A -20.000,E1 +7.737,E3 +110372.585,E4 +0.000} C_DIS
LIN {X -167.493,Y +1147.157,Z +0.000,A -20.000,E1 +16.195,E3 +110397.024,E4 +0.000} C_DIS
LIN {X -173.235,Y +1142.221,Z +0.000,A -20.000,E1 +22.930,E3 +110414.326,E4 +0.000} C_DIS
LIN {X -181.123,Y +1133.734,Z +0.000,A -20.000,E1 +30.868,E3 +110435.082,E4 +0.000} C_DIS
LIN {X -189.654,Y +1120.856,Z +0.000,A -20.000,E1 +39.018,E3 +110457.096,E4 +0.000} C_DIS
LIN {X -195.246,Y +1107.046,Z +0.000,A -20.000,E1 +44.515,E3 +110474.998,E4 +0.000} C_DIS
LIN {X -198.051,Y +1092.368,Z +0.000,A -20.000,E1 +47.947,E3 +110491.524,E4 +0.000} C_DIS
LIN {X -198.143,Y +1081.370,Z +0.000,A -19.806,E1 +49.153,E3 +110503.385,E4 +0.000} C_DIS
LIN {X -197.177,Y +1073.569,Z +0.000,A -17.356,E1 +49.162,E3 +110511.969,E4 +0.000} C_DIS
LIN {X -195.448,Y +1066.139,Z +0.000,A -12.154,E1 +48.512,E3 +110520.564,E4 +0.000} C_DIS
LIN {X -193.346,Y +1058.941,Z +0.000,A -7.133,E1 +47.724,E3 +110529.444,E4 +0.000} C_DIS
LIN {X -191.781,Y +1050.839,Z +0.000,A -3.715,E1 +47.274,E3 +110539.777,E4 +0.000} C_DIS
LIN {X -190.795,Y +1039.355,Z +0.000,A -0.983,E1 +46.842,E3 +110554.437,E4 +0.000} C_DIS
LIN {X -190.395,Y +1028.856,Z +0.000,A -0.089,E1 +46.598,E3 +110567.831,E4 +0.000} C_DIS
LIN {X -190.239,Y +1018.851,Z +0.000,A -0.004,E1 +46.529,E3 +110580.599,E4 +0.000} C_DIS
LIN {X -190.161,Y +1004.975,Z +0.000,A +0.000,E1 +46.506,E3 +110598.313,E4 +0.000} C_DIS
LIN {X -190.142,Y +412.853,Z +0.000,A +0.000,E1 +46.501,E3 +111354.519,E4 +0.000} C_DIS
LIN {X -190.147,Y +401.077,Z +0.000,A +0.000,E1 +46.499,E3 +111369.560,E4 +0.000} C_DIS
LIN {X -190.159,Y +390.929,Z +0.000,A +0.000,E1 +46.494,E3 +111382.526,E4 +0.000} C_DIS
LIN {X -190.174,Y +383.973,Z +0.000,A +0.000,E1 +46.484,E3 +111391.419,E4 +0.000} C_DIS
LIN {X -190.200,Y +373.815,Z +0.000,A +0.000,E1 +46.448,E3 +111404.424,E4 +0.000} C_DIS
LIN {X -190.154,Y +361.003,Z +0.000,A +0.000,E1 +46.303,E3 +111420.918,E4 +0.000} C_DIS
LIN {X -189.772,Y +350.660,Z +0.000,A +0.049,E1 +45.996,E3 +111434.457,E4 +0.000} C_DIS
LIN {X -189.325,Y +346.917,Z +0.000,A +0.243,E1 +45.771,E3 +111439.526,E4 +0.000} C_DIS
LIN {X -188.196,Y +342.754,Z +0.000,A +1.966,E1 +45.249,E3 +111445.534,E4 +0.000} C_DIS
LIN {X -185.199,Y +337.023,Z +0.000,A +6.630,E1 +43.793,E3 +111454.908,E4 +0.000} C_DIS
LIN {X -181.141,Y +331.596,Z +0.000,A +12.274,E1 +41.569,E3 +111465.468,E4 +0.000} C_DIS
LIN {X -176.762,Y +326.804,Z +0.000,A +17.560,E1 +38.898,E3 +111476.892,E4 +0.000} C_DIS
LIN {X -172.184,Y +322.578,Z +0.000,A +19.859,E1 +36.197,E3 +111489.622,E4 +0.000} C_DIS
LIN {X -165.998,Y +317.874,Z +0.000,A +20.000,E1 +32.027,E3 +111509.380,E4 +0.000} C_DIS
LIN {X -160.137,Y +314.334,Z +0.000,A +20.000,E1 +26.368,E3 +111533.749,E4 +0.000} C_DIS
LIN {X -155.624,Y +312.245,Z +0.000,A +20.000,E1 +19.506,E3 +111562.425,E4 +0.000} C_DIS
LIN {X -153.557,Y +311.879,Z +0.000,A +20.000,E1 +11.113,E3 +111598.180,E4 +0.000} C_DIS
LIN {X -155.320,Y +313.348,Z +0.000,A +20.000,E1 +3.401,E3 +111631.364,E4 +0.000} C_DIS
LIN {X -160.005,Y +315.804,Z +0.000,A +20.000,E1 -4.720,E3 +111661.742,E4 +0.000} C_DIS
LIN {X -164.504,Y +318.255,Z +0.000,A +20.000,E1 -10.663,E3 +111681.111,E4 +0.000} C_DIS
LIN {X -170.340,Y +322.684,Z +0.000,A +20.000,E1 -17.457,E3 +111701.143,E4 +0.000} C_DIS
LIN {X -175.568,Y +329.106,Z +0.000,A +20.000,E1 -24.747,E3 +111718.377,E4 +0.000} C_DIS
LIN {X -184.074,Y +340.065,Z +0.000,A +20.000,E1 -33.664,E3 +111741.317,E4 +0.000} C_DIS
LIN {X -190.779,Y +351.388,Z +0.000,A +20.000,E1 -40.083,E3 +111759.095,E4 +0.000} C_DIS
LIN {X -195.254,Y +362.955,Z +0.000,A +20.000,E1 -44.515,E3 +111773.848,E4 +0.000} C_DIS
LIN {X -197.754,Y +374.780,Z +0.000,A +20.000,E1 -47.450,E3 +111787.270,E4 +0.000} C_DIS
LIN {X -198.310,Y +383.215,Z +0.000,A +19.956,E1 -48.698,E3 +111796.394,E4 +0.000} C_DIS
LIN {X -197.912,Y +391.275,Z +0.000,A +18.601,E1 -49.158,E3 +111805.112,E4 +0.000} C_DIS
LIN {X -196.679,Y +398.944,Z +0.000,A +13.989,E1 -48.784,E3 +111813.666,E4 +0.000} C_DIS
LIN {X -194.742,Y +406.288,Z +0.000,A +8.476,E1 -48.001,E3 +111822.349,E4 +0.000} C_DIS
LIN {X -192.748,Y +413.472,Z +0.000,A +3.905,E1 -47.267,E3 +111831.359,E4 +0.000} C_DIS
LIN {X -191.781,Y +419.162,Z +0.000,A +1.739,E1 -46.975,E3 +111838.627,E4 +0.000} C_DIS
LIN {X -190.795,Y +430.646,Z +0.000,A +0.152,E1 -46.707,E3 +111853.288,E4 +0.000} C_DIS
LIN {X -190.395,Y +441.145,Z +0.000,A +0.001,E1 -46.583,E3 +111866.681,E4 +0.000} C_DIS
LIN {X -190.239,Y +451.150,Z +0.000,A -0.000,E1 -46.528,E3 +111879.449,E4 +0.000} C_DIS
LIN {X -190.161,Y +465.026,Z +0.000,A -0.000,E1 -46.506,E3 +111897.164,E4 +0.000} C_DIS
LIN {X -190.142,Y +1057.148,Z +0.000,A -0.000,E1 -46.500,E3 +112653.370,E4 +0.000} C_DIS
LIN {X -190.147,Y +1068.924,Z +0.000,A -0.000,E1 -46.499,E3 +112668.411,E4 +0.000} C_DIS
LIN {X -190.159,Y +1079.072,Z +0.000,A -0.000,E1 -46.493,E3 +112681.376,E4 +0.000} C_DIS
LIN {X -190.174,Y +1086.028,Z +0.000,A -0.000,E1 -46.483,E3 +112690.270,E4 +0.000} C_DIS
LIN {X -190.200,Y +1096.186,Z +0.000,A -0.000,E1 -46.448,E3 +112703.274,E4 +0.000} C_DIS
LIN {X -190.154,Y +1108.998,Z +0.000,A -0.054,E1 -46.295,E3 +112719.769,E4 +0.000} C_DIS
LIN {X -189.772,Y +1119.341,Z +0.000,A -0.752,E1 -45.902,E3 +112733.307,E4 +0.000} C_DIS
LIN {X -189.097,Y +1124.276,Z +0.000,A -2.508,E1 -45.397,E3 +112740.039,E4 +0.000} C_DIS
LIN {X -187.410,Y +1129.069,Z +0.000,A -5.304,E1 -44.585,E3 +112747.212,E4 +0.000} C_DIS
LIN {X -183.899,Y +1134.873,Z +0.000,A -10.372,E1 -42.805,E3 +112757.218,E4 +0.000} C_DIS
LIN {X -179.711,Y +1140.065,Z +0.000,A -15.940,E1 -40.393,E3 +112768.004,E4 +0.000} C_DIS
LIN {X -176.763,Y +1143.197,Z +0.000,A -18.748,E1 -38.674,E3 +112775.742,E4 +0.000} C_DIS
LIN {X -172.185,Y +1147.423,Z +0.000,A -19.971,E1 -36.175,E3 +112788.472,E4 +0.000} C_DIS
LIN {X -165.999,Y +1152.127,Z +0.000,A -20.000,E1 -32.027,E3 +112808.230,E4 +0.000} C_DIS
LIN {X -160.138,Y +1155.667,Z +0.000,A -20.000,E1 -26.368,E3 +112832.600,E4 +0.000} C_DIS
LIN {X -155.625,Y +1157.756,Z +0.000,A -20.000,E1 -19.505,E3 +112861.276,E4 +0.000} C_DIS
LIN {X -153.552,Y +1158.113,Z +0.000,A -20.000,E1 -11.113,E3 +112897.027,E4 +0.000} C_DIS
LIN {X -156.311,Y +1155.540,Z +0.000,A -20.000,E1 -0.839,E3 +112940.387,E4 +0.000} C_DIS
LIN {X -161.281,Y +1151.851,Z +0.000,A -20.000,E1 +7.737,E3 +112970.286,E4 +0.000} C_DIS
LIN {X -167.493,Y +1147.157,Z +0.000,A -20.000,E1 +16.195,E3 +112994.725,E4 +0.000} C_DIS
LIN {X -173.235,Y +1142.221,Z +0.000,A -20.000,E1 +22.930,E3 +113012.027,E4 +0.000} C_DIS
LIN {X -181.123,Y +1133.734,Z +0.000,A -20.000,E1 +30.868,E3 +113032.783,E4 +0.000} C_DIS
LIN {X -189.654,Y +1120.856,Z +0.000,A -20.000,E1 +39.018,E3 +113054.797,E4 +0.000} C_DIS
LIN {X -195.246,Y +1107.046,Z +0.000,A -20.000,E1 +44.515,E3 +113072.699,E4 +0.000} C_DIS
LIN {X -198.051,Y +1092.368,Z +0.000,A -20.000,E1 +47.947,E3 +113089.225,E4 +0.000} C_DIS
LIN {X -198.143,Y +1081.370,Z +0.000,A -19.806,E1 +49.153,E3 +113101.086,E4 +0.000} C_DIS
LIN {X -197.177,Y +1073.569,Z +0.000,A -17.356,E1 +49.162,E3 +113109.670,E4 +0.000} C_DIS
LIN {X -195.448,Y +1066.139,Z +0.000,A -12.154,E1 +48.512,E3 +113118.265,E4 +0.000} C_DIS
LIN {X -193.346,Y +1058.941,Z +0.000,A -7.133,E1 +47.724,E3 +113127.145,E4 +0.000} C_DIS
LIN {X -191.781,Y +1050.839,Z +0.000,A -3.715,E1 +47.274,E3 +113137.478,E4 +0.000} C_DIS
LIN {X -190.795,Y +1039.355,Z +0.000,A -0.983,E1 +46.842,E3 +113152.138,E4 +0.000} C_DIS
LIN {X -190.395,Y +1028.856,Z +0.000,A -0.089,E1 +46.598,E3 +113165.532,E4 +0.000} C_DIS
LIN {X -190.239,Y +1018.851,Z +0.000,A -0.004,E1 +46.529,E3 +113178.300,E4 +0.000} C_DIS
LIN {X -190.161,Y +1004.975,Z +0.000,A +0.000,E1 +46.506,E3 +113196.014,E4 +0.000} C_DIS
LIN {X -190.142,Y +412.853,Z +0.000,A +0.000,E1 +46.501,E3 +113952.220,E4 +0.000} C_DIS
LIN {X -190.147,Y +401.077,Z +0.000,A +0.000,E1 +46.499,E3 +113967.261,E4 +0.000} C_DIS
LIN {X -190.159,Y +390.929,Z +0.000,A +0.000,E1 +46.494,E3 +113980.227,E4 +0.000} C_DIS
LIN {X -190.174,Y +383.973,Z +0.000,A +0.000,E1 +46.484,E3 +113989.120,E4 +0.000} C_DIS
LIN {X -190.200,Y +373.815,Z +0.000,A +0.000,E1 +46.448,E3 +114002.125,E4 +0.000} C_DIS
LIN {X -190.154,Y +361.003,Z +0.000,A +0.000,E1 +46.303,E3 +114018.619,E4 +0.000} C_DIS
LIN {X -189.772,Y +350.660,Z +0.000,A +0.049,E1 +45.996,E3 +114032.158,E4 +0.000} C_DIS
LIN {X -189.325,Y +346.917,Z +0.000,A +0.243,E1 +45.771,E3 +114037.227,E4 +0.000} C_DIS
LIN {X -188.196,Y +342.754,Z +0.000,A +1.966,E1 +45.249,E3 +114043.235,E4 +0.000} C_DIS
LIN {X -185.199,Y +337.023,Z +0.000,A +6.630,E1 +43.793,E3 +114052.609,E4 +0.000} C_DIS
LIN {X -181.141,Y +331.596,Z +0.000,A +12.274,E1 +41.569,E3 +114063.169,E4 +0.000} C_DIS
LIN {X -176.762,Y +326.804,Z +0.000,A +17.560,E1 +38.898,E3 +114074.593,E4 +0.000} C_DIS
LIN {X -172.184,Y +322.578,Z +0.000,A +19.859,E1 +36.197,E3 +114087.323,E4 +0.000} C_DIS
LIN {X -165.998,Y +317.874,Z +0.000,A +20.000,E1 +32.027,E3 +114107.081,E4 +0.000} C_DIS
LIN {X -160.137,Y +314.334,Z +0.000,A +20.000,E1 +26.368,E3 +114131.450,E4 +0.000} C_DIS
LIN {X -155.624,Y +312.245,Z +0.000,A +20.000,E1 +19.506,E3 +114160.126,E4 +0.000} C_DIS
LIN {X -153.557,Y +311.879,Z +0.000,A +20.000,E1 +11.113,E3 +114195.881,E4 +0.000} C_DIS
LIN {X -155.320,Y +313.348,Z +0.000,A +20.000,E1 +3.401,E3 +114229.065,E4 +0.000} C_DIS
LIN {X -160.005,Y +315.804,Z +0.000,A +20.000,E1 -4.720,E3 +114259.443,E4 +0.000} C_DIS
LIN {X -164.504,Y +318.255,Z +0.000,A +20.000,E1 -10.663,E3 +114278.812,E4 +0.000} C_DIS
LIN {X -170.340,Y +322.684,Z +0.000,A +20.000,E1 -17.457,E3 +114298.844,E4 +0.000} C_DIS
LIN {X -175.568,Y +329.106,Z +0.000,A +20.000,E1 -24.747,E3 +114316.078,E4 +0.000} C_DIS
LIN {X -184.074,Y +340.065,Z +0.000,A +20.000,E1 -33.664,E3 +114339.018,E4 +0.000} C_DIS
LIN {X -190.779,Y +351.388,Z +0.000,A +20.000,E1 -40.083,E3 +114356.796,E4 +0.000} C_DIS
LIN {X -195.254,Y +362.955,Z +0.000,A +20.000,E1 -44.515,E3 +114371.549,E4 +0.000} C_DIS
LIN {X -197.754,Y +374.780,Z +0.000,A +20.000,E1 -47.450,E3 +114384.971,E4 +0.000} C_DIS
LIN {X -198.310,Y +383.215,Z +0.000,A +19.956,E1 -48.698,E3 +114394.095,E4 +0.000} C_DIS
LIN {X -197.912,Y +391.275,Z +0.000,A +18.601,E1 -49.158,E3 +114402.813,E4 +0.000} C_DIS
LIN {X -196.679,Y +398.944,Z +0.000,A +13.989,E1 -48.784,E3 +114411.367,E4 +0.000} C_DIS
LIN {X -194.742,Y +406.288,Z +0.000,A +8.476,E1 -48.001,E3 +114420.050,E4 +0.000} C_DIS
LIN {X -192.748,Y +413.472,Z +0.000,A +3.905,E1 -47.267,E3 +114429.060,E4 +0.000} C_DIS
LIN {X -191.781,Y +419.162,Z +0.000,A +1.739,E1 -46.975,E3 +114436.328,E4 +0.000} C_DIS
LIN {X -190.795,Y +430.646,Z +0.000,A +0.152,E1 -46.707,E3 +114450.989,E4 +0.000} C_DIS
LIN {X -190.395,Y +441.145,Z +0.000,A +0.001,E1 -46.583,E3 +114464.382,E4 +0.000} C_DIS
LIN {X -190.239,Y +451.150,Z +0.000,A -0.000,E1 -46.528,E3 +114477.150,E4 +0.000} C_DIS
LIN {X -190.161,Y +465.026,Z +0.000,A -0.000,E1 -46.506,E3 +114494.865,E4 +0.000} C_DIS
LIN {X -190.142,Y +1057.148,Z +0.000,A -0.000,E1 -46.500,E3 +115251.071,E4 +0.000} C_DIS
LIN {X -190.147,Y +1068.924,Z +0.000,A -0.000,E1 -46.499,E3 +115266.112,E4 +0.000} C_DIS
LIN {X -190.159,Y +1079.072,Z +0.000,A -0.000,E1 -46.493,E3 +115279.077,E4 +0.000} C_DIS
LIN {X -190.174,Y +1086.028,Z +0.000,A -0.000,E1 -46.483,E3 +115287.971,E4 +0.000} C_DIS
LIN {X -190.200,Y +1096.186,Z +0.000,A -0.000,E1 -46.448,E3 +115300.975,E4 +0.000} C_DIS
LIN {X -190.154,Y +1108.998,Z +0.000,A -0.054,E1 -46.295,E3 +115317.470,E4 +0.000} C_DIS
LIN {X -189.772,Y +1119.341,Z +0.000,A -0.752,E1 -45.902,E3 +115331.008,E4 +0.000} C_DIS
LIN {X -189.097,Y +1124.276,Z +0.000,A -2.508,E1 -45.397,E3 +115337.740,E4 +0.000} C_DIS
LIN {X -187.410,Y +1129.069,Z +0.000,A -5.304,E1 -44.585,E3 +115344.913,E4 +0.000} C_DIS
LIN {X -183.899,Y +1134.873,Z +0.000,A -10.372,E1 -42.805,E3 +115354.919,E4 +0.000} C_DIS
LIN {X -179.711,Y +1140.065,Z +0.000,A -15.940,E1 -40.393,E3 +115365.705,E4 +0.000} C_DIS
LIN {X -176.763,Y +1143.197,Z +0.000,A -18.748,E1 -38.674,E3 +115373.443,E4 +0.000} C_DIS
LIN {X -172.185,Y +1147.423,Z +0.000,A -19.971,E1 -36.175,E3 +115386.173,E4 +0.000} C_DIS
LIN {X -165.999,Y +1152.127,Z +0.000,A -20.000,E1 -32.027,E3 +115405.931,E4 +0.000} C_DIS
LIN {X -160.138,Y +1155.667,Z +0.000,A -20.000,E1 -26.368,E3 +115430.301,E4 +0.000} C_DIS
LIN {X -155.625,Y +1157.756,Z +0.000,A -20.000,E1 -19.505,E3 +115458.977,E4 +0.000} C_DIS
LIN {X -153.552,Y +1158.113,Z +0.000,A -20.000,E1 -11.113,E3 +115494.728,E4 +0.000} C_DIS
LIN {X -156.311,Y +1155.540,Z +0.000,A -20.000,E1 -0.839,E3 +115538.088,E4 +0.000} C_DIS
LIN {X -161.281,Y +1151.851,Z +0.000,A -20.000,E1 +7.737,E3 +115567.987,E4 +0.000} C_DIS
LIN {X -167.493,Y +1147.157,Z +0.000,A -20.000,E1 +16.195,E3 +115592.426,E4 +0.000} C_DIS
LIN {X -173.235,Y +1142.221,Z +0.000,A -20.000,E1 +22.930,E3 +115609.728,E4 +0.000} C_DIS
LIN {X -181.123,Y +1133.734,Z +0.000,A -20.000,E1 +30.868,E3 +115630.484,E4 +0.000} C_DIS
LIN {X -189.654,Y +1120.856,Z +0.000,A -20.000,E1 +39.018,E3 +115652.498,E4 +0.000} C_DIS
LIN {X -195.246,Y +1107.046,Z +0.000,A -20.000,E1 +44.515,E3 +115670.400,E4 +0.000} C_DIS
LIN {X -198.051,Y +1092.368,Z +0.000,A -20.000,E1 +47.947,E3 +115686.926,E4 +0.000} C_DIS
LIN {X -198.143,Y +1081.370,Z +0.000,A -19.806,E1 +49.153,E3 +115698.787,E4 +0.000} C_DIS
LIN {X -197.177,Y +1073.569,Z +0.000,A -17.356,E1 +49.162,E3 +115707.371,E4 +0.000} C_DIS
LIN {X -195.448,Y +1066.139,Z +0.000,A -12.154,E1 +48.512,E3 +115715.966,E4 +0.000} C_DIS
LIN {X -193.346,Y +1058.941,Z +0.000,A -7.133,E1 +47.724,E3 +115724.846,E4 +0.000} C_DIS
LIN {X -191.781,Y +1050.839,Z +0.000,A -3.715,E1 +47.274,E3 +115735.179,E4 +0.000} C_DIS
LIN {X -190.795,Y +1039.355,Z +0.000,A -0.983,E1 +46.842,E3 +115749.839,E4 +0.000} C_DIS
LIN {X -190.395,Y +1028.856,Z +0.000,A -0.089,E1 +46.598,E3 +115763.233,E4 +0.000} C_DIS
LIN {X -190.239,Y +1018.851,Z +0.000,A -0.004,E1 +46.529,E3 +115776.001,E4 +0.000} C_DIS
LIN {X -190.161,Y +1004.975,Z +0.000,A +0.000,E1 +46.506,E3 +115793.715,E4 +0.000} C_DIS
LIN {X -190.142,Y +412.853,Z +0.000,A +0.000,E1 +46.501,E3 +116549.921,E4 +0.000} C_DIS
LIN {X -190.147,Y +401.077,Z +0.000,A +0.000,E1 +46.499,E3 +116564.962,E4 +0.000} C_DIS
LIN {X -190.159,Y +390.929,Z +0.000,A +0.000,E1 +46.494,E3 +116577.928,E4 +0.000} C_DIS
LIN {X -190.174,Y +383.973,Z +0.000,A +0.000,E1 +46.484,E3 +116586.821,E4 +0.000} C_DIS
LIN {X -190.200,Y +373.815,Z +0.000,A +0.000,E1 +46.448,E3 +116599.826,E4 +0.000} C_DIS
LIN {X -190.154,Y +361.003,Z +0.000,A +0.000,E1 +46.303,E3 +116616.320,E4 +0.000} C_DIS
LIN {X -189.772,Y +350.660,Z +0.000,A +0.049,E1 +45.996,E3 +116629.859,E4 +0.000} C_DIS
LIN {X -189.325,Y +346.917,Z +0.000,A +0.243,E1 +45.771,E3 +116634.928,E4 +0.000} C_DIS
LIN {X -188.196,Y +342.754,Z +0.000,A +1.966,E1 +45.249,E3 +116640.936,E4 +0.000} C_DIS
LIN {X -185.199,Y +337.023,Z +0.000,A +6.630,E1 +43.793,E3 +116650.310,E4 +0.000} C_DIS
LIN {X -181.141,Y +331.596,Z +0.000,A +12.274,E1 +41.569,E3 +116660.870,E4 +0.000} C_DIS
LIN {X -176.762,Y +326.804,Z +0.000,A +17.560,E1 +38.898,E3 +116672.294,E4 +0.000} C_DIS
LIN {X -172.184,Y +322.578,Z +0.000,A +19.859,E1 +36.197,E3 +116685.024,E4 +0.000} C_DIS
LIN {X -165.998,Y +317.874,Z +0.000,A +20.000,E1 +32.027,E3 +116704.782,E4 +0.000} C_DIS
LIN {X -160.137,Y +314.334,Z +0.000,A +20.000,E1 +26.368,E3 +116729.151,E4 +0.000} C_DIS
LIN {X -155.624,Y +312.245,Z +0.000,A +20.000,E1 +19.506,E3 +116757.827,E4 +0.000} C_DIS
LIN {X -153.557,Y +311.879,Z +0.000,A +20.000,E1 +11.113,E3 +116793.582,E4 +0.000} C_DIS
LIN {X -155.320,Y +313.348,Z +0.000,A +20.000,E1 +3.401,E3 +116826.766,E4 +0.000} C_DIS
LIN {X -160.005,Y +315.804,Z +0.000,A +20.000,E1 -4.720,E3 +116857.144,E4 +0.000} C_DIS
LIN {X -164.504,Y +318.255,Z +0.000,A +20.000,E1 -10.663,E3 +116876.513,E4 +0.000} C_DIS
LIN {X -170.340,Y +322.684,Z +0.000,A +20.000,E1 -17.457,E3 +116896.545,E4 +0.000} C_DIS
LIN {X -175.568,Y +329.106,Z +0.000,A +20.000,E1 -24.747,E3 +116913.779,E4 +0.000} C_DIS
LIN {X -184.074,Y +340.065,Z +0.000,A +20.000,E1 -33.664,E3 +116936.719,E4 +0.000} C_DIS
LIN {X -190.779,Y +351.388,Z +0.000,A +20.000,E1 -40.083,E3 +116954.497,E4 +0.000} C_DIS
LIN {X -195.254,Y +362.955,Z +0.000,A +20.000,E1 -44.515,E3 +116969.250,E4 +0.000} C_DIS
LIN {X -197.754,Y +374.780,Z +0.000,A +20.000,E1 -47.450,E3 +116982.672,E4 +0.000} C_DIS
LIN {X -198.310,Y +383.215,Z +0.000,A +19.956,E1 -48.698,E3 +116991.796,E4 +0.000} C_DIS
LIN {X -197.912,Y +391.275,Z +0.000,A +18.601,E1 -49.158,E3 +117000.514,E4 +0.000} C_DIS
LIN {X -196.679,Y +398.944,Z +0.000,A +13.989,E1 -48.784,E3 +117009.068,E4 +0.000} C_DIS
LIN {X -194.742,Y +406.288,Z +0.000,A +8.476,E1 -48.001,E3 +117017.751,E4 +0.000} C_DIS
LIN {X -192.748,Y +413.472,Z +0.000,A +3.905,E1 -47.267,E3 +117026.761,E4 +0.000} C_DIS
LIN {X -191.781,Y +419.162,Z +0.000,A +1.739,E1 -46.975,E3 +117034.029,E4 +0.000} C_DIS
LIN {X -190.795,Y +430.646,Z +0.000,A +0.152,E1 -46.707,E3 +117048.690,E4 +0.000} C_DIS
LIN {X -190.395,Y +441.145,Z +0.000,A +0.001,E1 -46.583,E3 +117062.083,E4 +0.000} C_DIS
LIN {X -190.239,Y +451.150,Z +0.000,A -0.000,E1 -46.528,E3 +117074.851,E4 +0.000} C_DIS
LIN {X -190.161,Y +465.026,Z +0.000,A -0.000,E1 -46.506,E3 +117092.566,E4 +0.000} C_DIS
LIN {X -190.142,Y +1057.148,Z +0.000,A -0.000,E1 -46.500,E3 +117848.772,E4 +0.000} C_DIS
LIN {X -190.147,Y +1068.924,Z +0.000,A -0.000,E1 -46.499,E3 +117863.813,E4 +0.000} C_DIS
LIN {X -190.159,Y +1079.072,Z +0.000,A -0.000,E1 -46.493,E3 +117876.778,E4 +0.000} C_DIS
LIN {X -190.174,Y +1086.028,Z +0.000,A -0.000,E1 -46.483,E3 +117885.672,E4 +0.000} C_DIS
LIN {X -190.200,Y +1096.186,Z +0.000,A -0.000,E1 -46.448,E3 +117898.676,E4 +0.000} C_DIS
LIN {X -190.154,Y +1108.998,Z +0.000,A -0.054,E1 -46.295,E3 +117915.171,E4 +0.000} C_DIS
LIN {X -189.772,Y +1119.341,Z +0.000,A -0.752,E1 -45.902,E3 +117928.709,E4 +0.000} C_DIS
LIN {X -189.097,Y +1124.276,Z +0.000,A -2.508,E1 -45.397,E3 +117935.441,E4 +0.000} C_DIS
LIN {X -187.410,Y +1129.069,Z +0.000,A -5.304,E1 -44.585,E3 +117942.614,E4 +0.000} C_DIS
LIN {X -183.899,Y +1134.873,Z +0.000,A -10.372,E1 -42.805,E3 +117952.620,E4 +0.000} C_DIS
LIN {X -179.711,Y +1140.065,Z +0.000,A -15.940,E1 -40.393,E3 +117963.406,E4 +0.000} C_DIS
LIN {X -176.763,Y +1143.197,Z +0.000,A -18.748,E1 -38.674,E3 +117971.144,E4 +0.000} C_DIS
LIN {X -172.185,Y +1147.423,Z +0.000,A -19.971,E1 -36.175,E3 +117983.874,E4 +0.000} C_DIS
LIN {X -165.999,Y +1152.127,Z +0.000,A -20.000,E1 -32.027,E3 +118003.632,E4 +0.000} C_DIS
LIN {X -160.138,Y +1155.667,Z +0.000,A -20.000,E1 -26.368,E3 +118028.002,E4 +0.000} C_DIS
LIN {X -155.625,Y +1157.756,Z +0.000,A -20.000,E1 -19.505,E3 +118056.678,E4 +0.000} C_DIS
LIN {X -153.552,Y +1158.113,Z +0.000,A -20.000,E1 -11.113,E3 +118092.429,E4 +0.000} C_DIS
LIN {X -156.311,Y +1155.540,Z +0.000,A -20.000,E1 -0.839,E3 +118135.789,E4 +0.000} C_DIS
LIN {X -161.281,Y +1151.851,Z +0.000,A -20.000,E1 +7.737,E3 +118165.688,E4 +0.000} C_DIS
LIN {X -167.493,Y +1147.157,Z +0.000,A -20.000,E1 +16.195,E3 +118190.127,E4 +0.000} C_DIS
LIN {X -173.235,Y +1142.221,Z +0.000,A -20.000,E1 +22.930,E3 +118207.429,E4 +0.000} C_DIS
LIN {X -181.123,Y +1133.734,Z +0.000,A -20.000,E1 +30.868,E3 +118228.185,E4 +0.000} C_DIS
LIN {X -189.654,Y +1120.856,Z +0.000,A -20.000,E1 +39.018,E3 +118250.199,E4 +0.000} C_DIS
LIN {X -195.246,Y +1107.046,Z +0.000,A -20.000,E1 +44.515,E3 +118268.101,E4 +0.000} C_DIS
LIN {X -198.051,Y +1092.368,Z +0.000,A -20.000,E1 +47.947,E3 +118284.627,E4 +0.000} C_DIS
LIN {X -198.143,Y +1081.370,Z +0.000,A -19.806,E1 +49.153,E3 +118296.488,E4 +0.000} C_DIS
LIN {X -197.177,Y +1073.569,Z +0.000,A -17.356,E1 +49.162,E3 +118305.072,E4 +0.000} C_DIS
LIN {X -195.448,Y +1066.139,Z +0.000,A -12.154,E1 +48.512,E3 +118313.667,E4 +0.000} C_DIS
LIN {X -193.346,Y +1058.941,Z +0.000,A -7.133,E1 +47.724,E3 +118322.547,E4 +0.000} C_DIS
LIN {X -191.781,Y +1050.839,Z +0.000,A -3.715,E1 +47.274,E3 +118332.880,E4 +0.000} C_DIS
LIN {X -190.795,Y +1039.355,Z +0.000,A -0.983,E1 +46.842,E3 +118347.540,E4 +0.000} C_DIS
LIN {X -190.395,Y +1028.856,Z +0.000,A -0.089,E1 +46.598,E3 +118360.934,E4 +0.000} C_DIS
LIN {X -190.239,Y +1018.851,Z +0.000,A -0.004,E1 +46.529,E3 +118373.702,E4 +0.000} C_DIS
LIN {X -190.161,Y +1004.975,Z +0.000,A +0.000,E1 +46.506,E3 +118391.416,E4 +0.000} C_DIS
LIN {X -190.142,Y +412.853,Z +0.000,A +0.000,E1 +46.501,E3 +119147.622,E4 +0.000} C_DIS
LIN {X -190.147,Y +401.077,Z +0.000,A +0.000,E1 +46.499,E3 +119162.663,E4 +0.000} C_DIS
LIN {X -190.159,Y +390.929,Z +0.000,A +0.000,E1 +46.494,E3 +119175.629,E4 +0.000} C_DIS
LIN {X -190.174,Y +383.973,Z +0.000,A +0.000,E1 +46.484,E3 +119184.522,E4 +0.000} C_DIS
LIN {X -190.200,Y +373.815,Z +0.000,A +0.000,E1 +46.448,E3 +119197.527,E4 +0.000} C_DIS
LIN {X -190.154,Y +361.003,Z +0.000,A +0.000,E1 +46.303,E3 +119214.021,E4 +0.000} C_DIS
LIN {X -189.772,Y +350.660,Z +0.000,A +0.049,E1 +45.996,E3 +119227.560,E4 +0.000} C_DIS
LIN {X -189.325,Y +346.917,Z +0.000,A +0.243,E1 +45.771,E3 +119232.629,E4 +0.000} C_DIS
LIN {X -188.196,Y +342.754,Z +0.000,A +1.966,E1 +45.249,E3 +119238.637,E4 +0.000} C_DIS
LIN {X -185.199,Y +337.023,Z +0.000,A +6.630,E1 +43.793,E3 +119248.011,E4 +0.000} C_DIS
LIN {X -181.141,Y +331.596,Z +0.000,A +12.274,E1 +41.569,E3 +119258.571,E4 +0.000} C_DIS
LIN {X -176.762,Y +326.804,Z +0.000,A +17.560,E1 +38.898,E3 +119269.995,E4 +0.000} C_DIS
LIN {X -172.184,Y +322.578,Z +0.000,A +19.859,E1 +36.197,E3 +119282.725,E4 +0.000} C_DIS
LIN {X -165.998,Y +317.874,Z +0.000,A +20.000,E1 +32.027,E3 +119302.483,E4 +0.000} C_DIS
LIN {X -160.137,Y +314.334,Z +0.000,A +20.000,E1 +26.368,E3 +119326.852,E4 +0.000} C_DIS
LIN {X -155.624,Y +312.245,Z +0.000,A +20.000,E1 +19.506,E3 +119355.528,E4 +0.000} C_DIS
LIN {X -153.557,Y +311.879,Z +0.000,A +20.000,E1 +11.113,E3 +119391.283,E4 +0.000} C_DIS
LIN {X -155.320,Y +313.348,Z +0.000,A +20.000,E1 +3.401,E3 +119424.467,E4 +0.000} C_DIS
LIN {X -160.005,Y +315.804,Z +0.000,A +20.000,E1 -4.720,E3 +119454.845,E4 +0.000} C_DIS
LIN {X -164.504,Y +318.255,Z +0.000,A +20.000,E1 -10.663,E3 +119474.214,E4 +0.000} C_DIS
LIN {X -170.340,Y +322.684,Z +0.000,A +20.000,E1 -17.457,E3 +119494.246,E4 +0.000} C_DIS
LIN {X -175.568,Y +329.106,Z +0.000,A +20.000,E1 -24.747,E3 +119511.480,E4 +0.000} C_DIS
LIN {X -184.074,Y +340.065,Z +0.000,A +20.000,E1 -33.664,E3 +119534.420,E4 +0.000} C_DIS
LIN {X -190.779,Y +351.388,Z +0.000,A +20.000,E1 -40.083,E3 +119552.198,E4 +0.000} C_DIS
LIN {X -195.254,Y +362.955,Z +0.000,A +20.000,E1 -44.515,E3 +119566.951,E4 +0.000} C_DIS
LIN {X -197.754,Y +374.780,Z +0.000,A +20.000,E1 -47.450,E3 +119580.373,E4 +0.000} C_DIS
LIN {X -198.310,Y +383.215,Z +0.000,A +19.956,E1 -48.698,E3 +119589.497,E4 +0.000} C_DIS
LIN {X -197.912,Y +391.275,Z +0.000,A +18.601,E1 -49.158,E3 +119598.215,E4 +0.000} C_DIS
LIN {X -196.679,Y +398.944,Z +0.000,A +13.989,E1 -48.784,E3 +119606.769,E4 +0.000} C_DIS
LIN {X -194.742,Y +406.288,Z +0.000,A +8.476,E1 -48.001,E3 +119615.452,E4 +0.000} C_DIS
LIN {X -192.748,Y +413.472,Z +0.000,A +3.905,E1 -47.267,E3 +119624.462,E4 +0.000} C_DIS
LIN {X -191.781,Y +419.162,Z +0.000,A +1.739,E1 -46.975,E3 +119631.730,E4 +0.000} C_DIS
LIN {X -190.795,Y +430.646,Z +0.000,A +0.152,E1 -46.707,E3 +119646.391,E4 +0.000} C_DIS
LIN {X -190.395,Y +441.145,Z +0.000,A +0.001,E1 -46.583,E3 +119659.784,E4 +0.000} C_DIS
LIN {X -190.239,Y +451.150,Z +0.000,A -0.000,E1 -46.528,E3 +119672.552,E4 +0.000} C_DIS
LIN {X -190.161,Y +465.026,Z +0.000,A -0.000,E1 -46.506,E3 +119690.267,E4 +0.000} C_DIS
LIN {X -190.142,Y +1057.148,Z +0.000,A -0.000,E1 -46.500,E3 +120446.473,E4 +0.000} C_DIS
LIN {X -190.147,Y +1068.924,Z +0.000,A -0.000,E1 -46.499,E3 +120461.514,E4 +0.000} C_DIS
LIN {X -190.159,Y +1079.072,Z +0.000,A -0.000,E1 -46.493,E3 +120474.479,E4 +0.000} C_DIS
LIN {X -190.174,Y +1086.028,Z +0.000,A -0.000,E1 -46.483,E3 +120483.373,E4 +0.000} C_DIS
LIN {X -190.200,Y +1096.186,Z +0.000,A -0.000,E1 -46.448,E3 +120496.377,E4 +0.000} C_DIS
LIN {X -190.154,Y +1108.998,Z +0.000,A -0.054,E1 -46.295,E3 +120512.872,E4 +0.000} C_DIS
LIN {X -189.772,Y +1119.341,Z +0.000,A -0.752,E1 -45.902,E3 +120526.410,E4 +0.000} C_DIS
LIN {X -189.097,Y +1124.276,Z +0.000,A -2.508,E1 -45.397,E3 +120533.142,E4 +0.000} C_DIS
LIN {X -187.410,Y +1129.069,Z +0.000,A -5.304,E1 -44.585,E3 +120540.315,E4 +0.000} C_DIS
LIN {X -183.899,Y +1134.873,Z +0.000,A -10.372,E1 -42.805,E3 +120550.321,E4 +0.000} C_DIS
LIN {X -179.711,Y +1140.065,Z +0.000,A -15.940,E1 -40.393,E3 +120561.107,E4 +0.000} C_DIS
LIN {X -176.763,Y +1143.197,Z +0.000,A -18.748,E1 -38.674,E3 +120568.845,E4 +0.000} C_DIS
LIN {X -172.185,Y +1147.423,Z +0.000,A -19.971,E1 -36.175,E3 +120581.575,E4 +0.000} C_DIS
LIN {X -165.999,Y +1152.127,Z +0.000,A -20.000,E1 -32.027,E3 +120601.333,E4 +0.000} C_DIS
LIN {X -160.138,Y +1155.667,Z +0.000,A -20.000,E1 -26.368,E3 +120625.703,E4 +0.000} C_DIS
LIN {X -155.625,Y +1157.756,Z +0.000,A -20.000,E1 -19.505,E3 +120654.379,E4 +0.000} C_DIS
LIN {X -153.552,Y +1158.113,Z +0.000,A -20.000,E1 -11.113,E3 +120690.130,E4 +0.000} C_DIS
LIN {X -156.311,Y +1155.540,Z +0.000,A -20.000,E1 -0.839,E3 +120733.490,E4 +0.000} C_DIS
LIN {X -161.281,Y +1151.851,Z +0.000,A -20.000,E1 +7.737,E3 +120763.389,E4 +0.000} C_DIS
LIN {X -167.493,Y +1147.157,Z +0.000,A -20.000,E1 +16.195,E3 +120787.828,E4 +0.000} C_DIS
LIN {X -173.235,Y +1142.221,Z +0.000,A -20.000,E1 +22.930,E3 +120805.130,E4 +0.000} C_DIS
LIN {X -181.123,Y +1133.734,Z +0.000,A -20.000,E1 +30.868,E3 +120825.886,E4 +0.000} C_DIS
LIN {X -189.654,Y +1120.856,Z +0.000,A -20.000,E1 +39.018,E3 +120847.900,E4 +0.000} C_DIS
LIN {X -195.246,Y +1107.046,Z +0.000,A -20.000,E1 +44.515,E3 +120865.802,E4 +0.000} C_DIS
LIN {X -198.051,Y +1092.368,Z +0.000,A -20.000,E1 +47.947,E3 +120882.328,E4 +0.000} C_DIS
LIN {X -198.143,Y +1081.370,Z +0.000,A -19.806,E1 +49.153,E3 +120894.189,E4 +0.000} C_DIS
LIN {X -197.177,Y +1073.569,Z +0.000,A -17.356,E1 +49.162,E3 +120902.773,E4 +0.000} C_DIS
LIN {X -195.448,Y +1066.139,Z +0.000,A -12.154,E1 +48.512,E3 +120911.368,E4 +0.000} C_DIS
LIN {X -193.346,Y +1058.941,Z +0.000,A -7.133,E1 +47.724,E3 +120920.248,E4 +0.000} C_DIS
LIN {X -191.781,Y +1050.839,Z +0.000,A -3.715,E1 +47.274,E3 +120930.581,E4 +0.000} C_DIS
LIN {X -190.795,Y +1039.355,Z +0.000,A -0.983,E1 +46.842,E3 +120945.241,E4 +0.000} C_DIS
LIN {X -190.395,Y +1028.856,Z +0.000,A -0.089,E1 +46.598,E3 +120958.635,E4 +0.000} C_DIS
LIN {X -190.239,Y +1018.851,Z +0.000,A -0.004,E1 +46.529,E3 +120971.403,E4 +0.000} C_DIS
LIN {X -190.161,Y +1004.975,Z +0.000,A +0.000,E1 +46.506,E3 +120989.117,E4 +0.000} C_DIS
LIN {X -190.142,Y +412.853,Z +0.000,A +0.000,E1 +46.501,E3 +121745.323,E4 +0.000} C_DIS
LIN {X -190.147,Y +401.077,Z +0.000,A +0.000,E1 +46.499,E3 +121760.364,E4 +0.000} C_DIS
LIN {X -190.159,Y +390.929,Z +0.000,A +0.000,E1 +46.494,E3 +121773.330,E4 +0.000} C_DIS
LIN {X -190.174,Y +383.973,Z +0.000,A +0.000,E1 +46.484,E3 +121782.223,E4 +0.000} C_DIS
LIN {X -190.200,Y +373.815,Z +0.000,A +0.000,E1 +46.448,E3 +121795.228,E4 +0.000} C_DIS
LIN {X -190.154,Y +361.003,Z +0.000,A +0.000,E1 +46.303,E3 +121811.722,E4 +0.000} C_DIS
LIN {X -189.772,Y +350.660,Z +0.000,A +0.049,E1 +45.996,E3 +121825.261,E4 +0.000} C_DIS
LIN {X -189.325,Y +346.917,Z +0.000,A +0.243,E1 +45.771,E3 +121830.330,E4 +0.000} C_DIS
LIN {X -188.196,Y +342.754,Z +0.000,A +1.966,E1 +45.249,E3 +121836.338,E4 +0.000} C_DIS
LIN {X -185.199,Y +337.023,Z +0.000,A +6.630,E1 +43.793,E3 +121845.712,E4 +0.000} C_DIS
LIN {X -181.141,Y +331.596,Z +0.000,A +12.274,E1 +41.569,E3 +121856.272,E4 +0.000} C_DIS
LIN {X -176.762,Y +326.804,Z +0.000,A +17.560,E1 +38.898,E3 +121867.696,E4 +0.000} C_DIS
LIN {X -172.184,Y +322.578,Z +0.000,A +19.859,E1 +36.197,E3 +121880.426,E4 +0.000} C_DIS
LIN {X -165.998,Y +317.874,Z +0.000,A +20.000,E1 +32.027,E3 +121900.184,E4 +0.000} C_DIS
LIN {X -160.137,Y +314.334,Z +0.000,A +20.000,E1 +26.368,E3 +121924.553,E4 +0.000} C_DIS
LIN {X -155.624,Y +312.245,Z +0.000,A +20.000,E1 +19.506,E3 +121953.229,E4 +0.000} C_DIS
LIN {X -153.557,Y +311.879,Z +0.000,A +20.000,E1 +11.113,E3 +121988.984,E4 +0.000} C_DIS
LIN {X -155.320,Y +313.348,Z +0.000,A +20.000,E1 +3.401,E3 +122022.168,E4 +0.000} C_DIS
LIN {X -160.005,Y +315.804,Z +0.000,A +20.000,E1 -4.720,E3 +122052.546,E4 +0.000} C_DIS
LIN {X -164.504,Y +318.255,Z +0.000,A +20.000,E1 -10.663,E3 +122071.915,E4 +0.000} C_DIS
LIN {X -170.340,Y +322.684,Z +0.000,A +20.000,E1 -17.457,E3 +122091.947,E4 +0.000} C_DIS
LIN {X -175.568,Y +329.106,Z +0.000,A +20.000,E1 -24.747,E3 +122109.181,E4 +0.000} C_DIS
LIN {X -184.074,Y +340.065,Z +0.000,A +20.000,E1 -33.664,E3 +122132.121,E4 +0.000} C_DIS
LIN {X -190.779,Y +351.388,Z +0.000,A +20.000,E1 -40.083,E3 +122149.899,E4 +0.000} C_DIS
LIN {X -195.254,Y +362.955,Z +0.000,A +20.000,E1 -44.515,E3 +122164.652,E4 +0.000} C_DIS
LIN {X -197.754,Y +374.780,Z +0.000,A +20.000,E1 -47.450,E3 +122178.074,E4 +0.000} C_DIS
LIN {X -198.310,Y +383.215,Z +0.000,A +19.956,E1 -48.698,E3 +122187.198,E4 +0.000} C_DIS
LIN {X -197.912,Y +391.275,Z +0.000,A +18.601,E1 -49.158,E3 +122195.916,E4 +0.000} C_DIS
LIN {X -196.679,Y +398.944,Z +0.000,A +13.989,E1 -48.784,E3 +122204.470,E4 +0.000} C_DIS
LIN {X -194.742,Y +406.288,Z +0.000,A +8.476,E1 -48.001,E3 +122213.153,E4 +0.000} C_DIS
LIN {X -192.748,Y +413.472,Z +0.000,A +3.905,E1 -47.267,E3 +122222.163,E4 +0.000} C_DIS
LIN {X -191.781,Y +419.162,Z +0.000,A +1.739,E1 -46.975,E3 +122229.431,E4 +0.000} C_DIS
LIN {X -190.795,Y +430.646,Z +0.000,A +0.152,E1 -46.707,E3 +122244.092,E4 +0.000} C_DIS
LIN {X -190.395,Y +441.145,Z +0.000,A +0.001,E1 -46.583,E3 +122257.485,E4 +0.000} C_DIS
LIN {X -190.239,Y +451.150,Z +0.000,A -0.000,E1 -46.528,E3 +122270.253,E4 +0.000} C_DIS
LIN {X -190.161,Y +465.026,Z +0.000,A -0.000,E1 -46.506,E3 +122287.968,E4 +0.000} C_DIS
LIN {X -190.142,Y +1057.148,Z +0.000,A -0.000,E1 -46.500,E3 +123044.174,E4 +0.000} C_DIS
LIN {X -190.147,Y +1068.924,Z +0.000,A -0.000,E1 -46.499,E3 +123059.215,E4 +0.000} C_DIS
LIN {X -190.159,Y +1079.072,Z +0.000,A -0.000,E1 -46.493,E3 +123072.180,E4 +0.000} C_DIS
LIN {X -190.174,Y +1086.028,Z +0.000,A -0.000,E1 -46.483,E3 +123081.074,E4 +0.000} C_DIS
LIN {X -190.200,Y +1096.186,Z +0.000,A -0.000,E1 -46.448,E3 +123094.078,E4 +0.000} C_DIS
LIN {X -190.154,Y +1108.998,Z +0.000,A -0.054,E1 -46.295,E3 +123110.573,E4 +0.000} C_DIS
LIN {X -189.772,Y +1119.341,Z +0.000,A -0.752,E1 -45.902,E3 +123124.111,E4 +0.000} C_DIS
LIN {X -189.097,Y +1124.276,Z +0.000,A -2.508,E1 -45.397,E3 +123130.843,E4 +0.000} C_DIS
LIN {X -187.410,Y +1129.069,Z +0.000,A -5.304,E1 -44.585,E3 +123138.016,E4 +0.000} C_DIS
LIN {X -183.899,Y +1134.873,Z +0.000,A -10.372,E1 -42.805,E3 +123148.022,E4 +0.000} C_DIS
LIN {X -179.711,Y +1140.065,Z +0.000,A -15.940,E1 -40.393,E3 +123158.808,E4 +0.000} C_DIS
LIN {X -176.763,Y +1143.197,Z +0.000,A -18.748,E1 -38.674,E3 +123166.546,E4 +0.000} C_DIS
LIN {X -172.185,Y +1147.423,Z +0.000,A -19.971,E1 -36.175,E3 +123179.276,E4 +0.000} C_DIS
LIN {X -165.999,Y +1152.127,Z +0.000,A -20.000,E1 -32.027,E3 +123199.034,E4 +0.000} C_DIS
LIN {X -160.138,Y +1155.667,Z +0.000,A -20.000,E1 -26.368,E3 +123223.404,E4 +0.000} C_DIS
LIN {X -155.625,Y +1157.756,Z +0.000,A -20.000,E1 -19.505,E3 +123252.080,E4 +0.000} C_DIS
LIN {X -153.552,Y +1158.113,Z +0.000,A -20.000,E1 -11.113,E3 +123287.831,E4 +0.000} C_DIS
LIN {X -156.311,Y +1155.540,Z +0.000,A -20.000,E1 -0.839,E3 +123331.191,E4 +0.000} C_DIS
LIN {X -161.281,Y +1151.851,Z +0.000,A -20.000,E1 +7.737,E3 +123361.090,E4 +0.000} C_DIS
LIN {X -167.493,Y +1147.157,Z +0.000,A -20.000,E1 +16.195,E3 +123385.529,E4 +0.000} C_DIS
LIN {X -173.235,Y +1142.221,Z +0.000,A -20.000,E1 +22.930,E3 +123402.831,E4 +0.000} C_DIS
LIN {X -181.123,Y +1133.734,Z +0.000,A -20.000,E1 +30.868,E3 +123423.587,E4 +0.000} C_DIS
LIN {X -189.654,Y +1120.856,Z +0.000,A -20.000,E1 +39.018,E3 +123445.601,E4 +0.000} C_DIS
LIN {X -195.246,Y +1107.046,Z +0.000,A -20.000,E1 +44.515,E3 +123463.503,E4 +0.000} C_DIS
LIN {X -198.051,Y +1092.368,Z +0.000,A -20.000,E1 +47.947,E3 +123480.029,E4 +0.000} C_DIS
LIN {X -198.143,Y +1081.370,Z +0.000,A -19.806,E1 +49.153,E3 +123491.890,E4 +0.000} C_DIS
LIN {X -197.177,Y +1073.569,Z +0.000,A -17.356,E1 +49.162,E3 +123500.474,E4 +0.000} C_DIS
LIN {X -195.448,Y +1066.139,Z +0.000,A -12.154,E1 +48.512,E3 +123509.069,E4 +0.000} C_DIS
LIN {X -193.346,Y +1058.941,Z +0.000,A -7.133,E1 +47.724,E3 +123517.949,E4 +0.000} C_DIS
LIN {X -191.781,Y +1050.839,Z +0.000,A -3.715,E1 +47.274,E3 +123528.282,E4 +0.000} C_DIS
LIN {X -190.795,Y +1039.355,Z +0.000,A -0.983,E1 +46.842,E3 +123542.942,E4 +0.000} C_DIS
LIN {X -190.395,Y +1028.856,Z +0.000,A -0.089,E1 +46.598,E3 +123556.336,E4 +0.000} C_DIS
LIN {X -190.239,Y +1018.851,Z +0.000,A -0.004,E1 +46.529,E3 +123569.104,E4 +0.000} C_DIS
LIN {X -190.161,Y +1004.975,Z +0.000,A +0.000,E1 +46.506,E3 +123586.818,E4 +0.000} C_DIS
LIN {X -190.142,Y +412.853,Z +0.000,A +0.000,E1 +46.501,E3 +124343.024,E4 +0.000} C_DIS
LIN {X -190.147,Y +401.077,Z +0.000,A +0.000,E1 +46.499,E3 +124358.065,E4 +0.000} C_DIS
LIN {X -190.159,Y +390.929,Z +0.000,A +0.000,E1 +46.494,E3 +124371.031,E4 +0.000} C_DIS
LIN {X -190.174,Y +383.973,Z +0.000,A +0.000,E1 +46.484,E3 +124379.924,E4 +0.000} C_DIS
LIN {X -190.200,Y +373.815,Z +0.000,A +0.000,E1 +46.448,E3 +124392.929,E4 +0.000} C_DIS
LIN {X -190.154,Y +361.003,Z +0.000,A +0.000,E1 +46.303,E3 +124409.423,E4 +0.000} C_DIS
LIN {X -189.772,Y +350.660,Z +0.000,A +0.049,E1 +45.996,E3 +124422.962,E4 +0.000} C_DIS
LIN {X -189.325,Y +346.917,Z +0.000,A +0.243,E1 +45.771,E3 +124428.031,E4 +0.000} C_DIS
LIN {X -188.196,Y +342.754,Z +0.000,A +1.966,E1 +45.249,E3 +124434.039,E4 +0.000} C_DIS
LIN {X -185.199,Y +337.023,Z +0.000,A +6.630,E1 +43.793,E3 +124443.413,E4 +0.000} C_DIS
LIN {X -181.141,Y +331.596,Z +0.000,A +12.274,E1 +41.569,E3 +124453.973,E4 +0.000} C_DIS
LIN {X -176.762,Y +326.804,Z +0.000,A +17.560,E1 +38.898,E3 +124465.397,E4 +0.000} C_DIS
LIN {X -172.184,Y +322.578,Z +0.000,A +19.859,E1 +36.197,E3 +124478.127,E4 +0.000} C_DIS
LIN {X -165.998,Y +317.874,Z +0.000,A +20.000,E1 +32.027,E3 +124497.885,E4 +0.000} C_DIS
LIN {X -160.137,Y +314.334,Z +0.000,A +20.000,E1 +26.368,E3 +124522.254,E4 +0.000} C_DIS
LIN {X -155.624,Y +312.245,Z +0.000,A +20.000,E1 +19.506,E3 +124550.930,E4 +0.000} C_DIS
LIN {X -153.557,Y +311.879,Z +0.000,A +20.000,E1 +11.113,E3 +124586.685,E4 +0.000} C_DIS
LIN {X -155.320,Y +313.348,Z +0.000,A +20.000,E1 +3.401,E3 +124619.869,E4 +0.000} C_DIS
LIN {X -160.005,Y +315.804,Z +0.000,A +20.000,E1 -4.720,E3 +124650.247,E4 +0.000} C_DIS
LIN {X -164.504,Y +318.255,Z +0.000,A +20.000,E1 -10.663,E3 +124669.616,E4 +0.000} C_DIS
LIN {X -170.340,Y +322.684,Z +0.000,A +20.000,E1 -17.457,E3 +124689.648,E4 +0.000} C_DIS
LIN {X -175.568,Y +329.106,Z +0.000,A +20.000,E1 -24.747,E3 +124706.882,E4 +0.000} C_DIS
LIN {X -184.074,Y +340.065,Z +0.000,A +20.000,E1 -33.664,E3 +124729.822,E4 +0.000} C_DIS
LIN {X -190.779,Y +351.388,Z +0.000,A +20.000,E1 -40.083,E3 +124747.600,E4 +0.000} C_DIS
LIN {X -195.254,Y +362.955,Z +0.000,A +20.000,E1 -44.515,E3 +124762.353,E4 +0.000} C_DIS
LIN {X -197.754,Y +374.780,Z +0.000,A +20.000,E1 -47.450,E3 +124775.775,E4 +0.000} C_DIS
LIN {X -198.310,Y +383.215,Z +0.000,A +19.956,E1 -48.698,E3 +124784.899,E4 +0.000} C_DIS
LIN {X -197.912,Y +391.275,Z +0.000,A +18.601,E1 -49.158,E3 +124793.617,E4 +0.000} C_DIS
LIN {X -196.679,Y +398.944,Z +0.000,A +13.989,E1 -48.784,E3 +124802.171,E4 +0.000} C_DIS
LIN {X -194.742,Y +406.288,Z +0.000,A +8.476,E1 -48.001,E3 +124810.854,E4 +0.000} C_DIS
LIN {X -192.748,Y +413.472,Z +0.000,A +3.905,E1 -47.267,E3 +124819.864,E4 +0.000} C_DIS
LIN {X -191.781,Y +419.162,Z +0.000,A +1.739,E1 -46.975,E3 +124827.132,E4 +0.000} C_DIS
LIN {X -190.795,Y +430.646,Z +0.000,A +0.152,E1 -46.707,E3 +124841.793,E4 +0.000} C_DIS
LIN {X -190.395,Y +441.145,Z +0.000,A +0.001,E1 -46.583,E3 +124855.186,E4 +0.000} C_DIS
LIN {X -190.239,Y +451.150,Z +0.000,A -0.000,E1 -46.528,E3 +124867.954,E4 +0.000} C_DIS
LIN {X -190.161,Y +465.026,Z +0.000,A -0.000,E1 -46.506,E3 +124885.669,E4 +0.000} C_DIS
LIN {X -190.142,Y +1057.148,Z +0.000,A -0.000,E1 -46.500,E3 +125641.875,E4 +0.000} C_DIS
LIN {X -190.147,Y +1068.924,Z +0.000,A -0.000,E1 -46.499,E3 +125656.916,E4 +0.000} C_DIS
LIN {X -190.159,Y +1079.072,Z +0.000,A -0.000,E1 -46.493,E3 +125669.881,E4 +0.000} C_DIS
LIN {X -190.174,Y +1086.028,Z +0.000,A -0.000,E1 -46.483,E3 +125678.775,E4 +0.000} C_DIS
LIN {X -190.200,Y +1096.186,Z +0.000,A -0.000,E1 -46.448,E3 +125691.779,E4 +0.000} C_DIS
LIN {X -190.154,Y +1108.998,Z +0.000,A -0.054,E1 -46.295,E3 +125708.274,E4 +0.000} C_DIS
LIN {X -189.772,Y +1119.341,Z +0.000,A -0.752,E1 -45.902,E3 +125721.812,E4 +0.000} C_DIS
LIN {X -189.097,Y +1124.276,Z +0.000,A -2.508,E1 -45.397,E3 +125728.544,E4 +0.000} C_DIS
LIN {X -187.410,Y +1129.069,Z +0.000,A -5.304,E1 -44.585,E3 +125735.717,E4 +0.000} C_DIS
LIN {X -183.899,Y +1134.873,Z +0.000,A -10.372,E1 -42.805,E3 +125745.723,E4 +0.000} C_DIS
LIN {X -179.711,Y +1140.065,Z +0.000,A -15.940,E1 -40.393,E3 +125756.509,E4 +0.000} C_DIS
LIN {X -176.763,Y +1143.197,Z +0.000,A -18.748,E1 -38.674,E3 +125764.247,E4 +0.000} C_DIS
LIN {X -172.185,Y +1147.423,Z +0.000,A -19.971,E1 -36.175,E3 +125776.977,E4 +0.000} C_DIS
LIN {X -165.999,Y +1152.127,Z +0.000,A -20.000,E1 -32.027,E3 +125796.735,E4 +0.000} C_DIS
LIN {X -160.138,Y +1155.667,Z +0.000,A -20.000,E1 -26.368,E3 +125821.105,E4 +0.000} C_DIS
LIN {X -155.625,Y +1157.756,Z +0.000,A -20.000,E1 -19.505,E3 +125849.781,E4 +0.000} C_DIS
LIN {X -153.552,Y +1158.113,Z +0.000,A -20.000,E1 -11.113,E3 +125885.532,E4 +0.000} C_DIS
LIN {X -156.311,Y +1155.540,Z +0.000,A -20.000,E1 -0.839,E3 +125928.892,E4 +0.000} C_DIS
LIN {X -161.281,Y +1151.851,Z +0.000,A -20.000,E1 +7.737,E3 +125958.791,E4 +0.000} C_DIS
LIN {X -167.493,Y +1147.157,Z +0.000,A -20.000,E1 +16.195,E3 +125983.230,E4 +0.000} C_DIS
